END_VAR
VAR (* helpers for the ST form of the networks *)
	_t186 : BOOL;
	_t180 : BOOL;
END_VAR
(*-------------------------------------------------------------------------------------------------ПЛАНОВАЯ ПЕРЕЗАГРУЗКА МОДЕМА*)
IF MODEM_PLANOVUY_REBOOT THEN
	TIMER_DAY(IN:=TRUE, PT:=REAL_TO_TIME(TIME_PLANOVAYA_REBBOT_MODEM*60000) );
	IF TIMER_DAY.ET=TIMER_DAY.PT AND (STEP_MAIN=10 OR STEP_MAIN=520)   THEN
		IF STEP_MAIN=10 THEN
			STEP_MAIN:=600;
			TIMER_DAY(IN:=FALSE, PT:=T#0s );
			TIMER_DAY;
		END_IF
		IF STEP_MAIN=520 THEN
			STEP_MAIN:=700;
			TIMER_DAY(IN:=FALSE, PT:=T#0s );
			TIMER_DAY;
		END_IF
	END_IF
ELSE
	TIMER_DAY(IN:=FALSE, PT:=T#0s );
	TIMER_DAY;
END_IF
(*-----------------------------------------------ПЛАНОВАЯ МОДЕМА ЕСЛИ СЕРВЕР НЕ ОТВЕТИЛ БОЛЬШЕ 10 МИНУТ (НАПРИМЕР)*)
IF MODEM_WATCH_DOG THEN
	TIMER_SEND_OK(IN:=TRUE, PT:=REAL_TO_TIME(TIME_WATCH_DOG*1000));
	IF TIMER_SEND_OK.ET=TIMER_SEND_OK.PT AND (STEP_MAIN=10 OR STEP_MAIN=520)   THEN
		IF STEP_MAIN=10 THEN
			STEP_MAIN:=600;
			TIMER_SEND_OK(IN:=FALSE, PT:=T#0s );
			TIMER_SEND_OK;
		END_IF
		IF STEP_MAIN=520 THEN
			STEP_MAIN:=700;
			TIMER_SEND_OK(IN:=FALSE, PT:=T#0s );
			TIMER_SEND_OK;
		END_IF
	END_IF


	FIND_TIMER_SEND_OK:=FIND(OTVET, STRING_SEND_OK);
	IF FIND_TIMER_SEND_OK<>0 THEN
		TIMER_SEND_OK(IN:=FALSE, PT:=T#0s );
		TIMER_SEND_OK;
	END_IF
ELSE
	TIMER_SEND_OK(IN:=FALSE, PT:=T#0s );
	TIMER_SEND_OK;
END_IF

(*--------------------------------------------------------------------------------------------------ПЕРЕЗАГРУЗКА МОДЕМА С КНОПКИ*)
IF REBOOT_MODEM_SP_307 THEN
	IF STEP_MAIN=10 THEN
		STEP_MAIN:=600;
		TIMER_DAY(IN:=FALSE, PT:=T#0s );
		TIMER_DAY;
	END_IF
	IF STEP_MAIN=520 THEN
		STEP_MAIN:=700;
		TIMER_DAY(IN:=FALSE, PT:=T#0s );
		TIMER_DAY;
	END_IF
	REBOOT_MODEM_SP_307:=FALSE;
END_IF
(*--------------------------------------------------------------------------------СЛУШАЕМ ПОРТ, ЗАПИСЫВАЕМ ЗНАЧЕНИЯ В ОТВЕТ*)
P:=GetByte(0);
OTVET:=CONCAT(OTVET,RBDATA_TO_STRING(p));
IF LEN(OTVET)>255 THEN
	OTVET:='';
END_IF

(*-----------------------------------------------------------------------------------------------------------ПЕРЕЗАГРУЗКА С КНОПКИ'*)
IF REBOOT_MODEM_SP_307
THEN
	STEP_MAIN:=600;
	REBOOT_MODEM_SP_307:=FALSE;
	TIMER_REBOOT(IN:=FALSE, PT:=T#0s );
	TIMER_REBOOT;
END_IF

(*----------------------------------------------------------------------------------------------------------------ТЕСТ ОТПРАВКИ СМС'*)
IF TEST_OTPRAVKI_SMS_SP_307
THEN
	STEP_MAIN:=500;
	TEST_OTPRAVKI_SMS_SP_307:=FALSE;
	TIMER_REBOOT(IN:=FALSE, PT:=T#0s );
	TIMER_REBOOT;
END_IF
(*------------------------------------------------------------------ПЕРЕЗАГРУЗКА ПО КОЛИЧЕСТВУ ПОПЫТОК С ОТВЕТОМ ERROR'*)
IF POPUTKA>500 AND STEP_MAIN=10
THEN
	STEP_MAIN:=600;
	TIMER_REBOOT(IN:=FALSE, PT:=T#0s );
	TIMER_REBOOT;
END_IF
(*--------------------------------------------------------------------------ПЕРЕЗАГРУЗКА ПО КОЛИЧЕСТВУ ПОПЫТОК ПО ВРЕМЕНИ*)
IF POPUTKA_PO_VREMENI>6 AND STEP_MAIN=10
THEN
	STEP_MAIN:=600;
	TIMER_REBOOT(IN:=FALSE, PT:=T#0s );
	TIMER_REBOOT;
END_IF
(*------------------------------------------------------------------ПЕРЕЗАГРУЗКА ПО КОЛИЧЕСТВУ ПОПЫТОК С ОТВЕТОМ ERROR'*)
IF POPUTKA_AVARIA>400 AND STEP_MAIN=520
THEN
	STEP_MAIN:=700;
	TIMER_REBOOT(IN:=FALSE, PT:=T#0s );
	TIMER_REBOOT;
END_IF
(*-------------------------------------------------------------------------ПЕРЕЗАГРУЗКА ПО КОЛИЧЕСТВУ ПОПЫТОК ПО ВРЕМЕНИ*)
IF POPUTKA_PO_VREMENI_AVARIA>6 AND STEP_MAIN=520
THEN
	STEP_MAIN:=700;
	TIMER_REBOOT(IN:=FALSE, PT:=T#0s );
	TIMER_REBOOT;
END_IF
(*-------------------------------------------------------------------------------------------------------------ОТПРАВКА СМС АВАРИИ*)
MODEM_SOOBSHENIE_AVARIA;
	IF AVAR_SMS AND STEP_MAIN=10 AND PUSK_SP_307 THEN
		STEP_MAIN:=500;
	END_IF
(*-------------------------------------------------------------------------------------------------ОСНОВНОЙ ЦИКЛ РАБОТЫ МОДЕМА*)
CASE STEP_MAIN OF
0:
	TIMER_REBOOT(IN:=FALSE, PT:=T#0s );
	TIMER_REBOOT;
	MODEM1_ON:=TRUE;
	TIMER_ZADERGKA_OTPRAVKI_SOOBSHENIY(IN:=FALSE, PT:=T#0s );
	TIMER_ZADERGKA_OTPRAVKI_SOOBSHENIY;
	STEP_MAIN:=10;
(*---------------------------------------------------------------------------------------------------ОТПРАВКА СООБЩЕНИЙ ПО GPRS*)
10:
	MODEM_GPRS;
(*---------------------------------------------------------------------------------------------------------ОТПРАВКА АВАРИЙ ПО СМС*)
500:
	SMS_MODEM_1:=0;
	POPUTKA_AVARIA:=0;
	POPUTKA_PO_VREMENI_AVARIA:=0;
	OTVET:='';
	STEP_AVARIA:=0;
	STEP_INTO:=0;
	TIMER_ZADERGKA_OTPRAVKI_SOOBSHENIY(IN:=FALSE, PT:=T#0s );
	TIMER_ZADERGKA_OTPRAVKI_SOOBSHENIY;
	STEP_MAIN:=520;
520:
	MODEM_SMS_AVARIA;
(*--------------------------------------------------------------------------------------------------------------ПЕРЕЗАГРУЗКА МОДЕМА*)
600:
	MODEM1_ON:=FALSE;
	TIMER_REBOOT(IN:=TRUE, PT:=t#2S );
	IF TIMER_REBOOT.ET=TIMER_REBOOT.PT THEN
		STEP_MAIN:=601;
	END_IF
601:
	POPUTKA:=0;
	POPUTKA_PO_VREMENI:=0;
	REBOOT:=REBOOT+1;
	OTVET:='';
	STEP_MAIN:=0;
	STEP_MODEM:=0;
	STEP_INTO:=0;
(*-------------------------------------------------------------------------------------ПЕРЕЗАГРУЗКА МОДЕМА БЕЗ СБРОСА АВАРИИ*)
700:
	MODEM1_ON:=FALSE;
	TIMER_REBOOT(IN:=TRUE, PT:=t#2S );
	IF TIMER_REBOOT.ET=TIMER_REBOOT.PT THEN
		STEP_MAIN:=701;
	END_IF
701:
	POPUTKA:=0;
	POPUTKA_PO_VREMENI:=0;
	POPUTKA_AVARIA:=0;
	POPUTKA_PO_VREMENI_AVARIA:=0;
	REBOOT:=REBOOT+1;
	OTVET:='';
	STEP_MODEM:=0;
	STEP_AVARIA:=0;
	STEP_INTO:=0;
	POPUTKA_POSLE_REBOOT:=POPUTKA_POSLE_REBOOT+1;
	IF POPUTKA_POSLE_REBOOT>=2 THEN
		STEP_MAIN:=0;
		POPUTKA_POSLE_REBOOT:=0;
	ELSE
		STEP_MAIN:=500;
	END_IF
END_CASE
END_PROGRAM
ACTION COMMAND_AT_CGATT:
(*-----------------------------AT+CGATT? ПРОВЕРКА РЕГИСТРАЦИИ В СЕТИ ЕСЛИ 1 ТО ПЕРЕСКАКИВАЕМ ПОДКЛЮЧЕНИЕ GPRS*)
CASE STEP_INTO OF
		0:
			STR_OK:='';
			STR_ERROR:='';
			OTVET:='';
			COMMAND:='';
			STEP_INTO:=1;
			TIMER_OTVET(IN:=FALSE, PT:=T#0s );
			TIMER_OTVET;
			PAUSA(IN:=FALSE, PT:=T#0s );
			PAUSA;
		1:
			COMMAND:='AT+CGATT?';(*<-------------------------------------------------------------------------------AT-КОМАНДА*)
			STR_OK:='+CGATT: 1$R$N$R$NOK'; (*<------------------------------------------------------------ПРАВИЛЬНЫЙ ОТВЕТ*)
			STR_ERROR:='+CGATT: 0$R$N$R$NOK'; (*<-----------------------------------------------------НЕПРАВИЛЬНЫЙ ОТВЕТ*)
			COMMAND:=CONCAT(COMMAND,'$R$N');
			SetByte(0,COMMAND,LEN(COMMAND));
			STEP_INTO:=2;
		2:
			FIND_OK:=FIND(OTVET, STR_OK);
			FIND_ERROR:=FIND(OTVET, STR_ERROR);

			IF FIND_OK<>0 THEN
				PAUSA(IN:=TRUE, PT:=ZADERGKA_PEREHODA );
				IF PAUSA.ET=PAUSA.PT THEN
					STEP_MODEM:=10;(*<-------------ПЕРЕХОД К СЛЕДУЮЩЕЙ КОМАНДЕ ЕСЛИ ОТВЕТ ПОЛОЖИТЕЛЬНЫЙ*)(*10*)
					STEP_INTO:=0;
					POPUTKA:=0;
					POPUTKA_PO_VREMENI:=0;
				END_IF
			END_IF
			IF FIND_ERROR<>0 THEN
				STEP_INTO:=0;
				STEP_MODEM:=1;
				POPUTKA:=POPUTKA+1;
			END_IF
			TIMER_OTVET(IN:=TRUE, PT:=OGIDANIE_OTVETA );
			IF TIMER_OTVET.ET=TIMER_OTVET.PT THEN
				STEP_INTO:=0;
				STEP_MODEM:=190;(*<-----------------------ПЕРЕХОДИМ НА ПОСЛЕДНИЙ ШАГ ЗАКРЫТИЕ СОЕДИНЕНИЯ*)(*190*)
				POPUTKA_PO_VREMENI:=POPUTKA_PO_VREMENI+1;
				TIMER_OTVET(IN:=FALSE, PT:=T#0s );
				TIMER_OTVET;
			END_IF
END_CASE
END_ACTION
ACTION COMMAND_AT_CIFSR:
(*---------------------------------------------------------------------------------------AT+CIFSR ПОДКЛЮЧАЕМ ЛОКАЛЬНЫЙ АДРЕС*)
CASE STEP_INTO OF
		0:
			STR_OK:='';
			STR_ERROR:='';
			OTVET:='';
			COMMAND:='';
			STEP_INTO:=1;
			TIMER_OTVET(IN:=FALSE, PT:=T#0s );
			TIMER_OTVET;
			PAUSA(IN:=FALSE, PT:=T#0s );
			PAUSA;
		1:
			COMMAND:='AT+CIFSR';(*<---------------------------------------------------------------------------------AT-КОМАНДА*)
			STR_OK:='.';(*<---------------------------------------------------------------------------------------ПРАВИЛЬНЫЙ ОТВЕТ*)
			STR_ERROR:='ERROR';(*<-------------------------------------------------------------------------НЕПРАВИЛЬНЫЙ ОТВЕТ*)
			COMMAND:=CONCAT(COMMAND,'$R$N');
			SetByte(0,COMMAND,LEN(COMMAND));
			STEP_INTO:=2;
		2:
			PAUSA(IN:=TRUE, PT:=T#1S ); (*-----------------------------------ЗАПУСКАЕМ ТАЙМЕР ПАУЗА ЧТО БЫ ПОЛУЧИТЬ IP*)
			IF PAUSA.ET=PAUSA.PT THEN
				STEP_INTO:=3;
			END_IF
		3:
			FIND_OK:=FIND(OTVET, STR_OK);
			FIND_ERROR:=FIND(OTVET, STR_ERROR);

			IF FIND_OK<>0 THEN
				STEP_MODEM:=60;(*<-----------------------------------------------------ПЕРЕХОД К СЛЕДУЮЩЕЙ КОМАНДЕ*)(*60*)
				STEP_INTO:=0;
				POPUTKA:=0;
				POPUTKA_PO_VREMENI:=0;
			END_IF
			IF FIND_ERROR<>0 THEN
				STEP_MODEM:=1;
				STEP_INTO:=0;
				POPUTKA:=POPUTKA+1;
			END_IF
			TIMER_OTVET(IN:=TRUE, PT:=OGIDANIE_OTVETA );
			IF TIMER_OTVET.ET=TIMER_OTVET.PT THEN
				STEP_INTO:=0;
				STEP_MODEM:=190;(*<-----------------------ПЕРЕХОДИМ НА ПОСЛЕДНИЙ ШАГ ЗАКРЫТИЕ СОЕДИНЕНИЯ*)(*190*)
				POPUTKA_PO_VREMENI:=POPUTKA_PO_VREMENI+1;
				TIMER_OTVET(IN:=FALSE, PT:=T#0s );
				TIMER_OTVET;
			END_IF
END_CASE
END_ACTION
ACTION COMMAND_AT_CIICR:
(*-------------------------------------------------------------------------------------------------------AT+CIICR ПОДКЛЮЧАЕМ GPRS*)
CASE STEP_INTO OF
		0:
			STR_OK:='';
			STR_ERROR:='';
			OTVET:='';
			COMMAND:='';
			STEP_INTO:=1;
			TIMER_OTVET(IN:=FALSE, PT:=T#0s );
			TIMER_OTVET;
			PAUSA(IN:=FALSE, PT:=T#0s );
			PAUSA;
		1:
			COMMAND:='AT+CIICR';(*<---------------------------------------------------------------------------------AT-КОМАНДА*)
			STR_OK:='OK';(*<------------------------------------------------------------------------------------ПРАВИЛЬНЫЙ ОТВЕТ*)
			STR_ERROR:='ERROR';(*<-------------------------------------------------------------------------НЕПРАВИЛЬНЫЙ ОТВЕТ*)
			COMMAND:=CONCAT(COMMAND,'$R$N');
			SetByte(0,COMMAND,LEN(COMMAND));
			STEP_INTO:=2;
		2:
			FIND_OK:=FIND(OTVET, STR_OK);
			FIND_ERROR:=FIND(OTVET, STR_ERROR);

			IF FIND_OK<>0 THEN
				PAUSA(IN:=TRUE, PT:=ZADERGKA_PEREHODA );
				IF PAUSA.ET=PAUSA.PT THEN
					STEP_MODEM:=50;(*<-------------------------------------------------ПЕРЕХОД К СЛЕДУЮЩЕЙ КОМАНДЕ*)(*50*)
					STEP_INTO:=0;
					POPUTKA:=0;
					POPUTKA_PO_VREMENI:=0;
				END_IF
			END_IF
			IF FIND_ERROR<>0 THEN
				STEP_INTO:=0;
				STEP_MODEM:=1;
				POPUTKA:=POPUTKA+1;
			END_IF
			TIMER_OTVET(IN:=TRUE, PT:=OGIDANIE_OTVETA );
			IF TIMER_OTVET.ET=TIMER_OTVET.PT THEN
				STEP_INTO:=0;
				STEP_MODEM:=190;(*<-----------------------ПЕРЕХОДИМ НА ПОСЛЕДНИЙ ШАГ ЗАКРЫТИЕ СОЕДИНЕНИЯ*)(*190*)
				POPUTKA_PO_VREMENI:=POPUTKA_PO_VREMENI+1;
				TIMER_OTVET(IN:=FALSE, PT:=T#0s );
				TIMER_OTVET;
			END_IF
END_CASE
END_ACTION
ACTION COMMAND_AT_CIPSEND_1:
(*---------------------------------------------------------------------------------------AT+CIPSEND ЗАПРОС НА ПЕРЕДАЧУ ДАННЫХ*)
CASE STEP_INTO OF
		0:
			STR_OK:='';
			STR_ERROR:='';
			OTVET:='';
			COMMAND:='';
			STEP_INTO:=1;
			TIMER_OTVET(IN:=FALSE, PT:=T#0s );
			TIMER_OTVET;
			PAUSA(IN:=FALSE, PT:=T#0s );
			PAUSA;
		1:
			COMMAND:='AT+CIPSEND';(*<------------------------------------------------------------------------------AT-КОМАНДА*)
			STR_OK:='>';(*<--------------------------------------------------------------------------------------ПРАВИЛЬНЫЙ ОТВЕТ*)
			STR_ERROR:='ERROR';(*<-------------------------------------------------------------------------НЕПРАВИЛЬНЫЙ ОТВЕТ*)
			COMMAND:=CONCAT(COMMAND,'$R$N');
			SetByte(0,COMMAND,LEN(COMMAND));
			STEP_INTO:=2;
		2:
			FIND_OK:=FIND(OTVET, STR_OK);
			FIND_ERROR:=FIND(OTVET, STR_ERROR);

			IF FIND_OK<>0 THEN
				PAUSA(IN:=TRUE, PT:=ZADERGKA_PEREHODA );
				IF PAUSA.ET=PAUSA.PT THEN
					STEP_MODEM:=80;(*<-------------------------------------------------ПЕРЕХОД К СЛЕДУЮЩЕЙ КОМАНДЕ*)(*80*)
					STEP_INTO:=0;
					POPUTKA:=0;
					POPUTKA_PO_VREMENI:=0;
					OTVET:='';
				END_IF
			END_IF
			IF FIND_ERROR<>0 THEN
				STEP_INTO:=0;
				STEP_MODEM:=1;
				POPUTKA:=POPUTKA+1;
			END_IF
			TIMER_OTVET(IN:=TRUE, PT:=OGIDANIE_OTVETA );
			IF TIMER_OTVET.ET=TIMER_OTVET.PT THEN
				STEP_INTO:=0;
				STEP_MODEM:=190;(*<-----------------------ПЕРЕХОДИМ НА ПОСЛЕДНИЙ ШАГ ЗАКРЫТИЕ СОЕДИНЕНИЯ*)(*190*)
				POPUTKA_PO_VREMENI:=POPUTKA_PO_VREMENI+1;
				TIMER_OTVET(IN:=FALSE, PT:=T#0s );
				TIMER_OTVET;
			END_IF
END_CASE
END_ACTION
ACTION COMMAND_AT_CIPSEND_2:
(*-----------------------------------------------------------------------------AT+CIPSEND ЗАПРОС НА ПЕРЕДАЧУ ДАННЫХ ПАКЕТ 2*)
CASE STEP_INTO OF
		0:
			STR_OK:='';
			STR_ERROR:='';
			OTVET:='';
			COMMAND:='';
			STEP_INTO:=1;
			TIMER_OTVET(IN:=FALSE, PT:=T#0s );
			TIMER_OTVET;
			PAUSA(IN:=FALSE, PT:=T#0s );
			PAUSA;
		1:
			COMMAND:='AT+CIPSEND';(*<------------------------------------------------------------------------------AT-КОМАНДА*)
			STR_OK:='>';(*<--------------------------------------------------------------------------------------ПРАВИЛЬНЫЙ ОТВЕТ*)
			STR_ERROR:='ERROR';(*<-------------------------------------------------------------------------НЕПРАВИЛЬНЫЙ ОТВЕТ*)
			COMMAND:=CONCAT(COMMAND,'$R$N');
			SetByte(0,COMMAND,LEN(COMMAND));
			STEP_INTO:=2;
		2:
			FIND_OK:=FIND(OTVET, STR_OK);
			FIND_ERROR:=FIND(OTVET, STR_ERROR);

			IF FIND_OK<>0 THEN
				PAUSA(IN:=TRUE, PT:=ZADERGKA_PEREHODA );
				IF PAUSA.ET=PAUSA.PT THEN
					STEP_MODEM:=100;(*<----------------------------------------------ПЕРЕХОД К СЛЕДУЮЩЕЙ КОМАНДЕ*)(*100*)
					STEP_INTO:=0;
					POPUTKA:=0;
					POPUTKA_PO_VREMENI:=0;
					OTVET:='';
				END_IF
			END_IF
			IF FIND_ERROR<>0 THEN
				STEP_INTO:=0;
				STEP_MODEM:=1;
				POPUTKA:=POPUTKA+1;
			END_IF
			TIMER_OTVET(IN:=TRUE, PT:=OGIDANIE_OTVETA );
			IF TIMER_OTVET.ET=TIMER_OTVET.PT THEN
				STEP_INTO:=0;
				STEP_MODEM:=190;(*<-----------------------ПЕРЕХОДИМ НА ПОСЛЕДНИЙ ШАГ ЗАКРЫТИЕ СОЕДИНЕНИЯ*)(*190*)
				POPUTKA_PO_VREMENI:=POPUTKA_PO_VREMENI+1;
				TIMER_OTVET(IN:=FALSE, PT:=T#0s );
				TIMER_OTVET;
			END_IF
END_CASE
END_ACTION
ACTION COMMAND_AT_CIPSEND_3:
(*-----------------------------------------------------------------------------AT+CIPSEND ЗАПРОС НА ПЕРЕДАЧУ ДАННЫХ ПАКЕТ 2*)
CASE STEP_INTO OF
		0:
			STR_OK:='';
			STR_ERROR:='';
			OTVET:='';
			COMMAND:='';
			STEP_INTO:=1;
			TIMER_OTVET(IN:=FALSE, PT:=T#0s );
			TIMER_OTVET;
			PAUSA(IN:=FALSE, PT:=T#0s );
			PAUSA;
		1:
			COMMAND:='AT+CIPSEND';(*<------------------------------------------------------------------------------AT-КОМАНДА*)
			STR_OK:='>';(*<--------------------------------------------------------------------------------------ПРАВИЛЬНЫЙ ОТВЕТ*)
			STR_ERROR:='ERROR';(*<-------------------------------------------------------------------------НЕПРАВИЛЬНЫЙ ОТВЕТ*)
			COMMAND:=CONCAT(COMMAND,'$R$N');
			SetByte(0,COMMAND,LEN(COMMAND));
			STEP_INTO:=2;
		2:
			FIND_OK:=FIND(OTVET, STR_OK);
			FIND_ERROR:=FIND(OTVET, STR_ERROR);

			IF FIND_OK<>0 THEN
				PAUSA(IN:=TRUE, PT:=ZADERGKA_PEREHODA );
				IF PAUSA.ET=PAUSA.PT THEN
					STEP_MODEM:=120;(*<----------------------------------------------ПЕРЕХОД К СЛЕДУЮЩЕЙ КОМАНДЕ*)(*120*)
					STEP_INTO:=0;
					POPUTKA:=0;
					POPUTKA_PO_VREMENI:=0;
					OTVET:='';
				END_IF
			END_IF
			IF FIND_ERROR<>0 THEN
				STEP_INTO:=0;
				STEP_MODEM:=1;
				POPUTKA:=POPUTKA+1;
			END_IF
			TIMER_OTVET(IN:=TRUE, PT:=OGIDANIE_OTVETA );
			IF TIMER_OTVET.ET=TIMER_OTVET.PT THEN
				STEP_INTO:=0;
				STEP_MODEM:=190;(*<-----------------------ПЕРЕХОДИМ НА ПОСЛЕДНИЙ ШАГ ЗАКРЫТИЕ СОЕДИНЕНИЯ*)(*190*)
				POPUTKA_PO_VREMENI:=POPUTKA_PO_VREMENI+1;
				TIMER_OTVET(IN:=FALSE, PT:=T#0s );
				TIMER_OTVET;
			END_IF
END_CASE
END_ACTION
ACTION COMMAND_AT_CIPSHUT:
(*----------------------------------------------------------------------------------AT+CIPSHUT СБРОСИТЬ ВСЕ TCP ПОДКЛЮЧЕНИЯ*)
CASE STEP_INTO OF
		0:
			STR_OK:='';
			STR_ERROR:='';
			OTVET:='';
			COMMAND:='';
			STEP_INTO:=1;
			TIMER_OTVET(IN:=FALSE, PT:=T#0s );
			TIMER_OTVET;
			PAUSA(IN:=FALSE, PT:=T#0s );
			PAUSA;
		1:
			COMMAND:='AT+CIPSHUT';(*<------------------------------------------------------------------------------AT-КОМАНДА*)
			STR_OK:='SHUT OK';(*<------------------------------------------------------------------------------ПРАВИЛЬНЫЙ ОТВЕТ*)
			STR_ERROR:='ERROR';(*<-------------------------------------------------------------------------НЕПРАВИЛЬНЫЙ ОТВЕТ*)
			COMMAND:=CONCAT(COMMAND,'$R$N');
			SetByte(0,COMMAND,LEN(COMMAND));
			STEP_INTO:=2;
		2:
			FIND_OK:=FIND(OTVET, STR_OK);
			FIND_ERROR:=FIND(OTVET, STR_ERROR);

			IF FIND_OK<>0 THEN
				PAUSA(IN:=TRUE, PT:=ZADERGKA_PEREHODA );
				IF PAUSA.ET=PAUSA.PT THEN
					STEP_MODEM:=30;(*<-------------------------------------------------ПЕРЕХОД К СЛЕДУЮЩЕЙ КОМАНДЕ*)(*30*)
					STEP_INTO:=0;
					POPUTKA:=0;
					POPUTKA_PO_VREMENI:=0;
				END_IF
			END_IF
			IF FIND_ERROR<>0 THEN
				STEP_INTO:=0;
				STEP_MODEM:=1;
				POPUTKA:=POPUTKA+1;
			END_IF
			TIMER_OTVET(IN:=TRUE, PT:=OGIDANIE_OTVETA );
			IF TIMER_OTVET.ET=TIMER_OTVET.PT THEN
				STEP_INTO:=0;
				STEP_MODEM:=190;(*<-----------------------ПЕРЕХОДИМ НА ПОСЛЕДНИЙ ШАГ ЗАКРЫТИЕ СОЕДИНЕНИЯ*)(*190*)
				POPUTKA_PO_VREMENI:=POPUTKA_PO_VREMENI+1;
				TIMER_OTVET(IN:=FALSE, PT:=T#0s );
				TIMER_OTVET;
			END_IF
END_CASE
END_ACTION
ACTION COMMAND_AT_CIPSTART:
(*-------------------------------------------------AT+CIPSTART="TCP","ingavino.teplotehnika68.ru",80 ПОДКЛЮЧАЕМСЯ К СЕРВЕРУ*)
CASE STEP_INTO OF
		0:
			STR_OK:='';
			STR_ERROR:='';
			OTVET:='';
			COMMAND:='';
			STEP_INTO:=1;
			TIMER_OTVET(IN:=FALSE, PT:=T#0s );
			TIMER_OTVET;
			PAUSA(IN:=FALSE, PT:=T#0s );
			PAUSA;
		1:
			COMMAND:='AT+CIPSTART="TCP","karaul.teplotehnika68.ru",80';(*<-----------------------------------AT-КОМАНДА*)
			STR_OK:='CONNECT OK';(*<-------------------------------------------------------------------------ПРАВИЛЬНЫЙ ОТВЕТ*)
			STR_ERROR:='ERROR';(*<-------------------------------------------------------------------------НЕПРАВИЛЬНЫЙ ОТВЕТ*)
			COMMAND:=CONCAT(COMMAND,'$R$N');
			SetByte(0,COMMAND,LEN(COMMAND));
			STEP_INTO:=2;
		2:
			FIND_OK:=FIND(OTVET, STR_OK);
			FIND_ERROR:=FIND(OTVET, STR_ERROR);
			IF FIND_OK<>0 THEN
				PAUSA(IN:=TRUE, PT:=ZADERGKA_PEREHODA );
				IF PAUSA.ET=PAUSA.PT THEN
					STEP_MODEM:=70;(*<-------------------------------------------------ПЕРЕХОД К СЛЕДУЮЩЕЙ КОМАНДЕ*)(*70*)
					STEP_INTO:=0;
					POPUTKA:=0;
					POPUTKA_PO_VREMENI:=0;
					OTVET:='';
				END_IF
			END_IF
			IF FIND_ERROR<>0 THEN
				STEP_MODEM:=1;
				STEP_INTO:=0;
				POPUTKA:=POPUTKA+1;
			END_IF
			TIMER_OTVET(IN:=TRUE, PT:=OGIDANIE_OTVETA );
			IF TIMER_OTVET.ET=TIMER_OTVET.PT THEN
				STEP_INTO:=0;
				STEP_MODEM:=190;(*<-----------------------ПЕРЕХОДИМ НА ПОСЛЕДНИЙ ШАГ ЗАКРЫТИЕ СОЕДИНЕНИЯ*)(*190*)
				POPUTKA_PO_VREMENI:=POPUTKA_PO_VREMENI+1;
				TIMER_OTVET(IN:=FALSE, PT:=T#0s );
				TIMER_OTVET;
			END_IF
END_CASE
END_ACTION
ACTION COMMAND_AT_CSTT:
(*--------------------------------------------------------------AT+CSTT="internet.mts.ru","mts","mts" НАСТРОЙКА ТОЧКИ ДОСТУПА*)
CASE STEP_INTO OF
		0:
			STR_OK:='';
			STR_ERROR:='';
			OTVET:='';
			COMMAND:='';
			STEP_INTO:=1;
			TIMER_OTVET(IN:=FALSE, PT:=T#0s );
			TIMER_OTVET;
			PAUSA(IN:=FALSE, PT:=T#0s );
			PAUSA;
		1:
			COMMAND:='AT+CSTT="internet.mts.ru","mts","mts"';(*<---------------------------------------------------AT-КОМАНДА*)
			STR_OK:='OK';(*<------------------------------------------------------------------------------------ПРАВИЛЬНЫЙ ОТВЕТ*)
			STR_ERROR:='ERROR';(*<-------------------------------------------------------------------------НЕПРАВИЛЬНЫЙ ОТВЕТ*)
			COMMAND:=CONCAT(COMMAND,'$R$N');
			SetByte(0,COMMAND,LEN(COMMAND));
			STEP_INTO:=2;
		2:
			FIND_OK:=FIND(OTVET, STR_OK);
			FIND_ERROR:=FIND(OTVET, STR_ERROR);

			IF FIND_OK<>0 THEN
				PAUSA(IN:=TRUE, PT:=ZADERGKA_PEREHODA );
				IF PAUSA.ET=PAUSA.PT THEN
					STEP_MODEM:=40;(*<-------------------------------------------------ПЕРЕХОД К СЛЕДУЮЩЕЙ КОМАНДЕ*)(*40*)
					STEP_INTO:=0;
					POPUTKA:=0;
					POPUTKA_PO_VREMENI:=0;
				END_IF
			END_IF
			IF FIND_ERROR<>0 THEN
				STEP_INTO:=0;
				STEP_MODEM:=1;
				POPUTKA:=POPUTKA+1;
			END_IF
			TIMER_OTVET(IN:=TRUE, PT:=OGIDANIE_OTVETA );
			IF TIMER_OTVET.ET=TIMER_OTVET.PT THEN
				STEP_INTO:=0;
				STEP_MODEM:=190;(*<-----------------------ПЕРЕХОДИМ НА ПОСЛЕДНИЙ ШАГ ЗАКРЫТИЕ СОЕДИНЕНИЯ*)(*190*)
				POPUTKA_PO_VREMENI:=POPUTKA_PO_VREMENI+1;
				TIMER_OTVET(IN:=FALSE, PT:=T#0s );
				TIMER_OTVET;
			END_IF
END_CASE
END_ACTION
ACTION COMMAND_ATE0:
(*---------------------------------------------------------------------------------------------------------------ATE0 ОТКЛЮЧИТЬ ЭХО*)
CASE STEP_INTO OF
		0:
			STR_OK:='';
			STR_ERROR:='';
			OTVET:='';
			COMMAND:='';
			STEP_INTO:=1;
			TIMER_OTVET(IN:=FALSE, PT:=T#0s );
			TIMER_OTVET;
			PAUSA(IN:=FALSE, PT:=T#0s );
			PAUSA;
		1:
			COMMAND:='ATE0';(*<--------------------------------------------------------------------------------------AT-КОМАНДА*)
			STR_OK:='OK';(*<------------------------------------------------------------------------------------ПРАВИЛЬНЫЙ ОТВЕТ*)
			STR_ERROR:='ERROR';(*<-------------------------------------------------------------------------НЕПРАВИЛЬНЫЙ ОТВЕТ*)
			COMMAND:=CONCAT(COMMAND,'$R$N');
			SetByte(0,COMMAND,LEN(COMMAND));
			STEP_INTO:=2;
		2:
			FIND_OK:=FIND(OTVET, STR_OK);
			FIND_ERROR:=FIND(OTVET, STR_ERROR);

			IF FIND_OK<>0 THEN
				PAUSA(IN:=TRUE, PT:=ZADERGKA_PEREHODA );
				IF PAUSA.ET=PAUSA.PT THEN
					STEP_MODEM:=20;(*<-------------------------------------------------ПЕРЕХОД К СЛЕДУЮЩЕЙ КОМАНДЕ*)(*20*)
					STEP_INTO:=0;
					POPUTKA:=0;
					POPUTKA_PO_VREMENI:=0;
				END_IF
			END_IF
			IF FIND_ERROR<>0 THEN
				STEP_INTO:=0;
				STEP_MODEM:=1;
				POPUTKA:=POPUTKA+1;
			END_IF
			TIMER_OTVET(IN:=TRUE, PT:=OGIDANIE_OTVETA );
			IF TIMER_OTVET.ET=TIMER_OTVET.PT THEN
				STEP_INTO:=0;
				STEP_MODEM:=190;(*<-----------------------ПЕРЕХОДИМ НА ПОСЛЕДНИЙ ШАГ ЗАКРЫТИЕ СОЕДИНЕНИЯ*)(*190*)
				POPUTKA_PO_VREMENI:=POPUTKA_PO_VREMENI+1;
				TIMER_OTVET(IN:=FALSE, PT:=T#0s );
				TIMER_OTVET;
			END_IF
END_CASE
END_ACTION
ACTION MODEM_FORMIROVANIE_SMS_AVARII:
IF (AVARIA_OBRUV_DATCHIKA_T1_SP_307 AND AVARIA_OBRUV_DATCHIKA_T2_SP_307 AND AVARIA_OBRUV_DATCHIKA_T3_SP_307
	AND AVARIA_OBRUV_DATCHIKA_T4_SP_307 AND AVARIA_OBRUV_DATCHIKA_T5_SP_307 AND AVARIA_OBRUV_DATCHIKA_T6_SP_307
		AND AVARIA_OBRUV_DATCHIKA_T7_SP_307 AND AVARIA_OBRUV_DATCHIKA_T8_SP_307)
	OR (AVARIA_OBRUV_DATCHIKA_P1_SP_307 AND AVARIA_OBRUV_DATCHIKA_P2_SP_307 AND AVARIA_OBRUV_DATCHIKA_P3_SP_307
		AND AVARIA_OBRUV_DATCHIKA_P4_SP_307 AND AVARIA_OBRUV_DATCHIKA_P5_SP_307 AND AVARIA_OBRUV_DATCHIKA_P6_SP_307
			AND AVARIA_OBRUV_DATCHIKA_P7_SP_307) THEN

			STRING_SEND:=CONCAT(STRING_SEND,'AVARIA MODUL 1$R$N');
ELSE
			IF AVARIA_SETEVOY_NASOS_1_SP_307 THEN
				STRING_SEND:=CONCAT(STRING_SEND,'SETEVOY NASOS 1$R$N');
			END_IF
			IF AVARIA_SETEVOY_NASOS_2_SP_307 THEN
				STRING_SEND:=CONCAT(STRING_SEND,'AVAR.SETEVOY NASOS 2$R$N');
			END_IF
			IF AVARIA_VNUTR_NASOS_1_SP_307 THEN
				STRING_SEND:=CONCAT(STRING_SEND,'VNUTREN NASOS 1$R$N');
			END_IF
			IF AVARIA_VNUTR_NASOS_2_SP_307 THEN
				STRING_SEND:=CONCAT(STRING_SEND,'VNUTREN NASOS 2$R$N');
			END_IF
			IF AVARIA_GVS_NASOS_1_SP_307 THEN
				STRING_SEND:=CONCAT(STRING_SEND,'NASOS GVS 1$R$N');
			END_IF
			IF AVARIA_GVS_NASOS_2_SP_307 THEN
				STRING_SEND:=CONCAT(STRING_SEND,'NASOS GVS 2$R$N');
			END_IF
			IF AVARIA_PODPITOCHNYU_NASOS_1_SP_307 THEN
				STRING_SEND:=CONCAT(STRING_SEND,'PODPIT NASOS 1$R$N');
			END_IF
			IF AVARIA_PODPITOCHNYU_NASOS_2_SP_307 THEN
				STRING_SEND:=CONCAT(STRING_SEND,'PODPIT NASOS 2$R$N');
			END_IF
			(*IF AVARIA_LETNIY_NASOS_SP_307 THEN
				STRING_SEND:=CONCAT(STRING_SEND,'NL ');
			END_IF*)
			IF AVARIA_GORELKA_1_SP_307 THEN
				STRING_SEND:=CONCAT(STRING_SEND,'GORELKA 1$R$N');
			END_IF
			IF AVARIA_GORELKA_2_SP_307 THEN
				STRING_SEND:=CONCAT(STRING_SEND,'GORELKA 2$R$N');
			END_IF
			IF AVARIA_GORELKA_3_SP_307 THEN
				STRING_SEND:=CONCAT(STRING_SEND,'GORELKA 3$R$N');
			END_IF
			IF PREDUPREGDENIE_VKLUCHITE_GORELKU_1_SP_307 THEN
				STRING_SEND:=CONCAT(STRING_SEND,'ON_G1 ');
			END_IF
			IF PREDUPREGDENIE_VKLUCHITE_GORELKU_2_SP_307 THEN
				STRING_SEND:=CONCAT(STRING_SEND,'ON_G2 ');
			END_IF
			IF AVARIA_PHASA_SP_307 THEN
				STRING_SEND:=CONCAT(STRING_SEND,'PHASA$R$N');
			END_IF
			IF AVARIA_FIRE_SP_307 THEN
				STRING_SEND:=CONCAT(STRING_SEND,'POJAR$R$N');
			END_IF
			IF AVARIA_GAZ_SP_307 THEN
				STRING_SEND:=CONCAT(STRING_SEND,'GAS$R$N');
			END_IF
			IF AVARIA_VUSOKOE_DAVLENIE_OTOPLENIYA_SP_307 THEN
				STRING_SEND:=CONCAT(STRING_SEND,'VUSOK DAVL OTOPL$R$N');
			END_IF
			IF AVARIA_NIZKOE_DAVLENIE_OTOPLENIYA_SP_307 THEN
				STRING_SEND:=CONCAT(STRING_SEND,'NIZKOE DAVL OTOP$R$N');
			END_IF
			IF AVARIA_VUSOKOE_DAVLENIE_GVS_SP_307 THEN
				STRING_SEND:=CONCAT(STRING_SEND,'VUSOK DAVL GVS$R$N');
			END_IF
			IF AVARIA_NIZKOE_DAVLENIE_GVS_SP_307 THEN
				STRING_SEND:=CONCAT(STRING_SEND,'NIZKOE DAVL GVS$R$N');
			END_IF
			IF AVARIA_OBRUV_DATCHIKA_T1_SP_307 THEN
				STRING_SEND:=CONCAT(STRING_SEND,'OBRUV DAT T1$R$N');
			END_IF
			IF AVARIA_OBRUV_DATCHIKA_T2_SP_307 THEN
				STRING_SEND:=CONCAT(STRING_SEND,'OBRUV DAT T2$R$N');
			END_IF
			IF AVARIA_OBRUV_DATCHIKA_T3_SP_307 THEN
				STRING_SEND:=CONCAT(STRING_SEND,'OBRUV DAT T3$R$N');
			END_IF
			IF AVARIA_OBRUV_DATCHIKA_T4_SP_307 THEN
				STRING_SEND:=CONCAT(STRING_SEND,'OBRUV DAT T4$R$N');
			END_IF
			IF AVARIA_OBRUV_DATCHIKA_T5_SP_307 THEN
				STRING_SEND:=CONCAT(STRING_SEND,'OBRUV DAT T5$R$N');
			END_IF
			IF AVARIA_OBRUV_DATCHIKA_T6_SP_307 THEN
				STRING_SEND:=CONCAT(STRING_SEND,'OBRUV DAT T6$R$N');
			END_IF
			IF AVARIA_OBRUV_DATCHIKA_T7_SP_307 THEN
				STRING_SEND:=CONCAT(STRING_SEND,'OBRUV DAT T7$R$N');
			END_IF
			IF AVARIA_OBRUV_DATCHIKA_T8_SP_307 THEN
				STRING_SEND:=CONCAT(STRING_SEND,'OBRUV DAT T8$R$N');
			END_IF
			IF AVARIA_OBRUV_DATCHIKA_P1_SP_307 THEN
				STRING_SEND:=CONCAT(STRING_SEND,'OBRUV DAT D1$R$N');
			END_IF
			IF AVARIA_OBRUV_DATCHIKA_P2_SP_307 THEN
				STRING_SEND:=CONCAT(STRING_SEND,'OBRUV DAT D2$R$N');
			END_IF
			IF AVARIA_OBRUV_DATCHIKA_P3_SP_307 THEN
				STRING_SEND:=CONCAT(STRING_SEND,'OBRUV DAT D3$R$N');
			END_IF
			IF AVARIA_OBRUV_DATCHIKA_P4_SP_307 THEN
				STRING_SEND:=CONCAT(STRING_SEND,'OBRUV DAT D4$R$N');
			END_IF
			IF AVARIA_OBRUV_DATCHIKA_P5_SP_307 THEN
				STRING_SEND:=CONCAT(STRING_SEND,'OBRUV DAT D5$R$N');
			END_IF
			IF AVARIA_OBRUV_DATCHIKA_P6_SP_307 THEN
				STRING_SEND:=CONCAT(STRING_SEND,'OBRUV DAT D6$R$N');
			END_IF
			IF AVARIA_OBRUV_DATCHIKA_P7_SP_307 THEN
				STRING_SEND:=CONCAT(STRING_SEND,'OBRUV DAT D7$R$N');
			END_IF
			IF AVARIA_VUSOKAYA_TEMPERATURA_KOTEL_1_SP_307 THEN
				STRING_SEND:=CONCAT(STRING_SEND,'VUSOK TEMPER KOTEL 1$R$N');
			END_IF
			IF AVARIA_VUSOKAYA_TEMPERATURA_KOTEL_2_SP_307 THEN
				STRING_SEND:=CONCAT(STRING_SEND,'VUSOK TEMPER KOTEL 2$R$N');
			END_IF
			IF AVARIA_VUSOKAYA_TEMPERATURA_KOTEL_3_SP_307 THEN
				STRING_SEND:=CONCAT(STRING_SEND,'VUSOK TEMPER KOTEL 3$R$N');
			END_IF
			IF AVARIA_NAKOPITELNUY_BAK_SP_307 THEN
				STRING_SEND:=CONCAT(STRING_SEND,'NAKOPITELNUY  BAK$R$N');
			END_IF
END_IF
END_ACTION
ACTION MODEM_GPRS:
CASE STEP_MODEM OF
(*--------------------------------------------------------------------------------------------ЗАДЕРЖКА ПОСЛЕ ВКЛЮЧЕНИЯ МОДЕМА*)
0:
	TIMER_ZADERGKA_OTPRAVKI_SOOBSHENIY(IN:=TRUE, PT:=TIME_ZADERGKA_OTPRAVKI_SOOBSHENIY );
	IF TIMER_ZADERGKA_OTPRAVKI_SOOBSHENIY.ET=TIMER_ZADERGKA_OTPRAVKI_SOOBSHENIY.PT THEN
		STEP_MODEM:=1;
	END_IF
(*-----------------------------AT+CGATT? ПРОВЕРКА РЕГИСТРАЦИИ В СЕТИ ЕСЛИ 1 ТО ПЕРЕСКАКИВАЕМ ПОДКЛЮЧЕНИЕ GPRS*)
1:
	COMMAND_AT_CGATT;
(*---------------------------------------------------------------------------------------------------------------ATE0 ОТКЛЮЧИТЬ ЭХО*)
10:
	COMMAND_ATE0;
(*----------------------------------------------------------------------------------AT+CIPSHUT СБРОСИТЬ ВСЕ TCP ПОДКЛЮЧЕНИЯ*)
20:
	COMMAND_AT_CIPSHUT;
(*--------------------------------------------------------------AT+CSTT="internet.mts.ru","mts","mts" НАСТРОЙКА ТОЧКИ ДОСТУПА*)
30:
	COMMAND_AT_CSTT;
(*-------------------------------------------------------------------------------------------------------AT+CIICR ПОДКЛЮЧАЕМ GPRS*)
40:
	COMMAND_AT_CIICR;
(*---------------------------------------------------------------------------------------AT+CIFSR ПОДКЛЮЧАЕМ ЛОКАЛЬНЫЙ АДРЕС*)
50:
	COMMAND_AT_CIFSR;
(*-------------------------------------------------AT+CIPSTART="TCP","ingavino.teplotehnika68.ru",80 ПОДКЛЮЧАЕМСЯ К СЕРВЕРУ*)
60:
	COMMAND_AT_CIPSTART;
(*-----------------------------------------------------------------------------AT+CIPSEND ЗАПРОС НА ПЕРЕДАЧУ ДАННЫХ ПАКЕТ 1*)
70:
	COMMAND_AT_CIPSEND_1;
(*---------------------------------------------------------------------------------------------------------ПЕРЕДАЧА ДАННЫХ ПАКЕТ 1*)
80:
	SEND_DATA_1;
(*-----------------------------------------------------------------------------AT+CIPSEND ЗАПРОС НА ПЕРЕДАЧУ ДАННЫХ ПАКЕТ 2*)
90:
	COMMAND_AT_CIPSEND_2;
(*---------------------------------------------------------------------------------------------------------ПЕРЕДАЧА ДАННЫХ ПАКЕТ 2*)
100:
	SEND_DATA_2;
(*-----------------------------------------------------------------------------AT+CIPSEND ЗАПРОС НА ПЕРЕДАЧУ ДАННЫХ ПАКЕТ 3*)
110:
	COMMAND_AT_CIPSEND_3;
(*---------------------------------------------------------------------------------------------------------ПЕРЕДАЧА ДАННЫХ ПАКЕТ 3*)
120:
	SEND_DATA_3;
(*----------------------------------------------------------------------------------------------------------------------------------------------------------AT+CIPSEND запрос на передачу данных--------*)


(*----------------------------------------------------------------------------------------------------------------------------------------------------------передача данных СТАТУС 2--------*)







(*----------------------------------------------------------------------------------------------------------------------------------------------------------AT+CIPSHUT СБРОСИТЬ ВСЕ TCP ПОДКЛЮЧЕНИЯ--------*)
190:
CASE STEP_INTO OF
		0:
			STR_OK:='';
			STR_ERROR:='';
			OTVET:='';
			COMMAND:='';
			STEP_INTO:=1;
			TIMER_OTVET(IN:=FALSE, PT:=T#0s );(*ОБНУЛЯЕМ ТАЙМЕР ОЖИДАНИЯ ОТВЕТА*)
			TIMER_OTVET;
			PAUSA(IN:=FALSE, PT:=T#0s );(*ОБНУЛЯЕМ ТАЙМЕР ПАУЗЫ ПЕРЕД СЛЕДУЮЩЕЙ КОМАНДОЙ*)
			PAUSA;
			SetByte(0,'$0D$0A$0D$0A$1A',6);
			SetByte(0,'$0D$0A$0D$0A$1B',6);
			SetByte(0,'$0D$0A',4);

		1:
			COMMAND:='AT+CIPSHUT';(*<---------------------AT-КОМАНДА*)
			STR_OK:='SHUT OK';(*<-----------------------------------ПРАВИЛЬНЫЙ ОТВЕТ*)
			STR_ERROR:='ERROR';(*<---------------------------НЕПРАВИЛЬНЫЙ ОТВЕТ*)
			COMMAND:=CONCAT(COMMAND,'$R$N');
			SetByte(0,COMMAND,LEN(COMMAND));
			STEP_INTO:=2;
		2:
			FIND_OK:=FIND(OTVET, STR_OK);
			FIND_ERROR:=FIND(OTVET, STR_ERROR);

			IF FIND_OK<>0 THEN
				PAUSA(IN:=TRUE, PT:=(*ZADERGKA_PEREHODA*)T#1s ); (*ТАЙМЕР ЗАДЕРЖКИ ПЕРЕХОДА*)
				IF PAUSA.ET=PAUSA.PT THEN
					STEP_MODEM:=60;(*<-----------------------------ПЕРЕХОД К СЛЕДУЮЩЕЙ КОМАНДЕ*)
					STEP_INTO:=0;
					POPUTKA:=0;
					POPUTKA_PO_VREMENI:=0;
				END_IF
			END_IF
			IF FIND_ERROR<>0 THEN
				STEP_INTO:=0;
				POPUTKA:=POPUTKA+1;
			END_IF
			TIMER_OTVET(IN:=TRUE, PT:=OGIDANIE_OTVETA ); (*ЗАПУСКАЕМ ТАЙМЕР ОТВЕТА ОТ МОДЕМА ПОКА 20 СЕК*)
			IF TIMER_OTVET.ET=TIMER_OTVET.PT THEN
				STEP_INTO:=0;
				POPUTKA_PO_VREMENI:=POPUTKA_PO_VREMENI+1;
				TIMER_OTVET(IN:=FALSE, PT:=T#0s );(*ОБНУЛЯЕМ ТАЙМЕР ОЖИДАНИЯ ОТВЕТА*)
				TIMER_OTVET;
			END_IF
	END_CASE

END_CASE
END_ACTION
ACTION MODEM_OTPRAVKA_SMS_AVARII_1:
CASE STEP_AVARIA OF
(*-----------------------------------------------------------------------------------------------------ЗАДЕРЖКА ВКЛЮЧЕНИЯ МОДЕМА*)
0:
	MODEM1_ON:=TRUE;
	TIMER_ZADERGKA_OTPRAVKI_SOOBSHENIY(IN:=TRUE, PT:=T#5s );
	IF TIMER_ZADERGKA_OTPRAVKI_SOOBSHENIY.ET=TIMER_ZADERGKA_OTPRAVKI_SOOBSHENIY.PT THEN
		SetByte(0,'$R$N$R$N$1A$R$N',6);
		TIMER_OTVET(IN:=FALSE, PT:=T#0s );
		TIMER_OTVET;
		NUMBER1:='';
		NUMBER2:='';
		NUMBER3:='';
		STEP_AVARIA:=1;
	END_IF
1:
	NUMBER1:=CONCAT(NUMBER1,'+7');
	NUMBER1:=CONCAT(NUMBER1,REAL_TO_STRING(TRUNC(TEL_KOD_1)));
	NUMBER1:=CONCAT(NUMBER1,REAL_TO_STRING(TRUNC(TEL_NOMER_1)));

	NUMBER2:=CONCAT(NUMBER2,'+7');
	NUMBER2:=CONCAT(NUMBER2,REAL_TO_STRING(TRUNC(TEL_KOD_2)));
	NUMBER2:=CONCAT(NUMBER2,REAL_TO_STRING(TRUNC(TEL_NOMER_2)));

	NUMBER3:=CONCAT(NUMBER3,'+7');
	NUMBER3:=CONCAT(NUMBER3,REAL_TO_STRING(TRUNC(TEL_KOD_3)));
	NUMBER3:=CONCAT(NUMBER3,REAL_TO_STRING(TRUNC(TEL_NOMER_3)));
	NUMBER:=NUMBER1;
	STEP_AVARIA:=10;
(*----------------------------------------------------------------------------------------------------------------ATE0 ОТКЛЮЧИТЬ ЭХО*)
10:
	SMS_ATE0;
(*-----------------------------AT+CGATT? ПРОВЕРКА РЕГИСТРАЦИИ В СЕТИ ЕСЛИ 1 ТО ПЕРЕСКАКИВАЕМ ПОДКЛЮЧЕНИЕ GPRS*)
20:
	SMS_AT_CGATT;
(*---------------------------------------------------------------------------------------AT+CIPSHUT СБРОСИТЬ ВСЕ ПОДКЛЮЧЕНИЯ*)
30:
	SMS_AT_CIPSHUT;
(*----------------------------------------------------------------------------------------AT+CMGF=1 ВКЛЮЧАЕМ ТЕКСТОВЫЙ РЕЖИМ*)
40:
	SMS_AT_CMGF_1;
(*--------------------------------------------------------------------------------------------------AT+CSCS="GSM" КОДИРОВКА GSM*)
50:
	SMS_AT_CSCS_GSM;
(*---------------------------------------------------------------------------------------------------AT+CMGS="ТЕЛЕФОННЫЙ НОМЕР"*)
60:
	SMS_AT_CMGS;
(*-------------------------------------------------------------------------------------------------------------------ПЕРЕДАЧА ДАННЫХ*)
70:
	SMS_SEND_DATA;
(*--------------------------------------------------------------------------------------------------------------ВЫХОД ИЗ РЕЖИМА СМС*)
75:
	SMS_MODEM_1:=SMS_MODEM_1+1;
	IF SMS_MODEM_1>KOLICESTVO_SOOBSHENIY*KOLICHESTVO_NOMEROV-1 THEN
		STEP_MAIN:=0;
		STEP_MODEM:=1;
		NUMBER:=NUMBER1;
		TEL:=1;
	ELSE
		STEP_AVARIA:=10;
		IF TEL=1 THEN
			NUMBER:=NUMBER1;
		END_IF
		IF TEL=2 THEN
			NUMBER:=NUMBER2;
		END_IF
		IF TEL=3 THEN
			NUMBER:=NUMBER3;
		END_IF
	END_IF
END_CASE
END_ACTION
ACTION MODEM_SMS_AVARIA:
MODEM_OTPRAVKA_SMS_AVARII_1;
END_ACTION
ACTION MODEM_SOOBSHENIE_AVARIA:
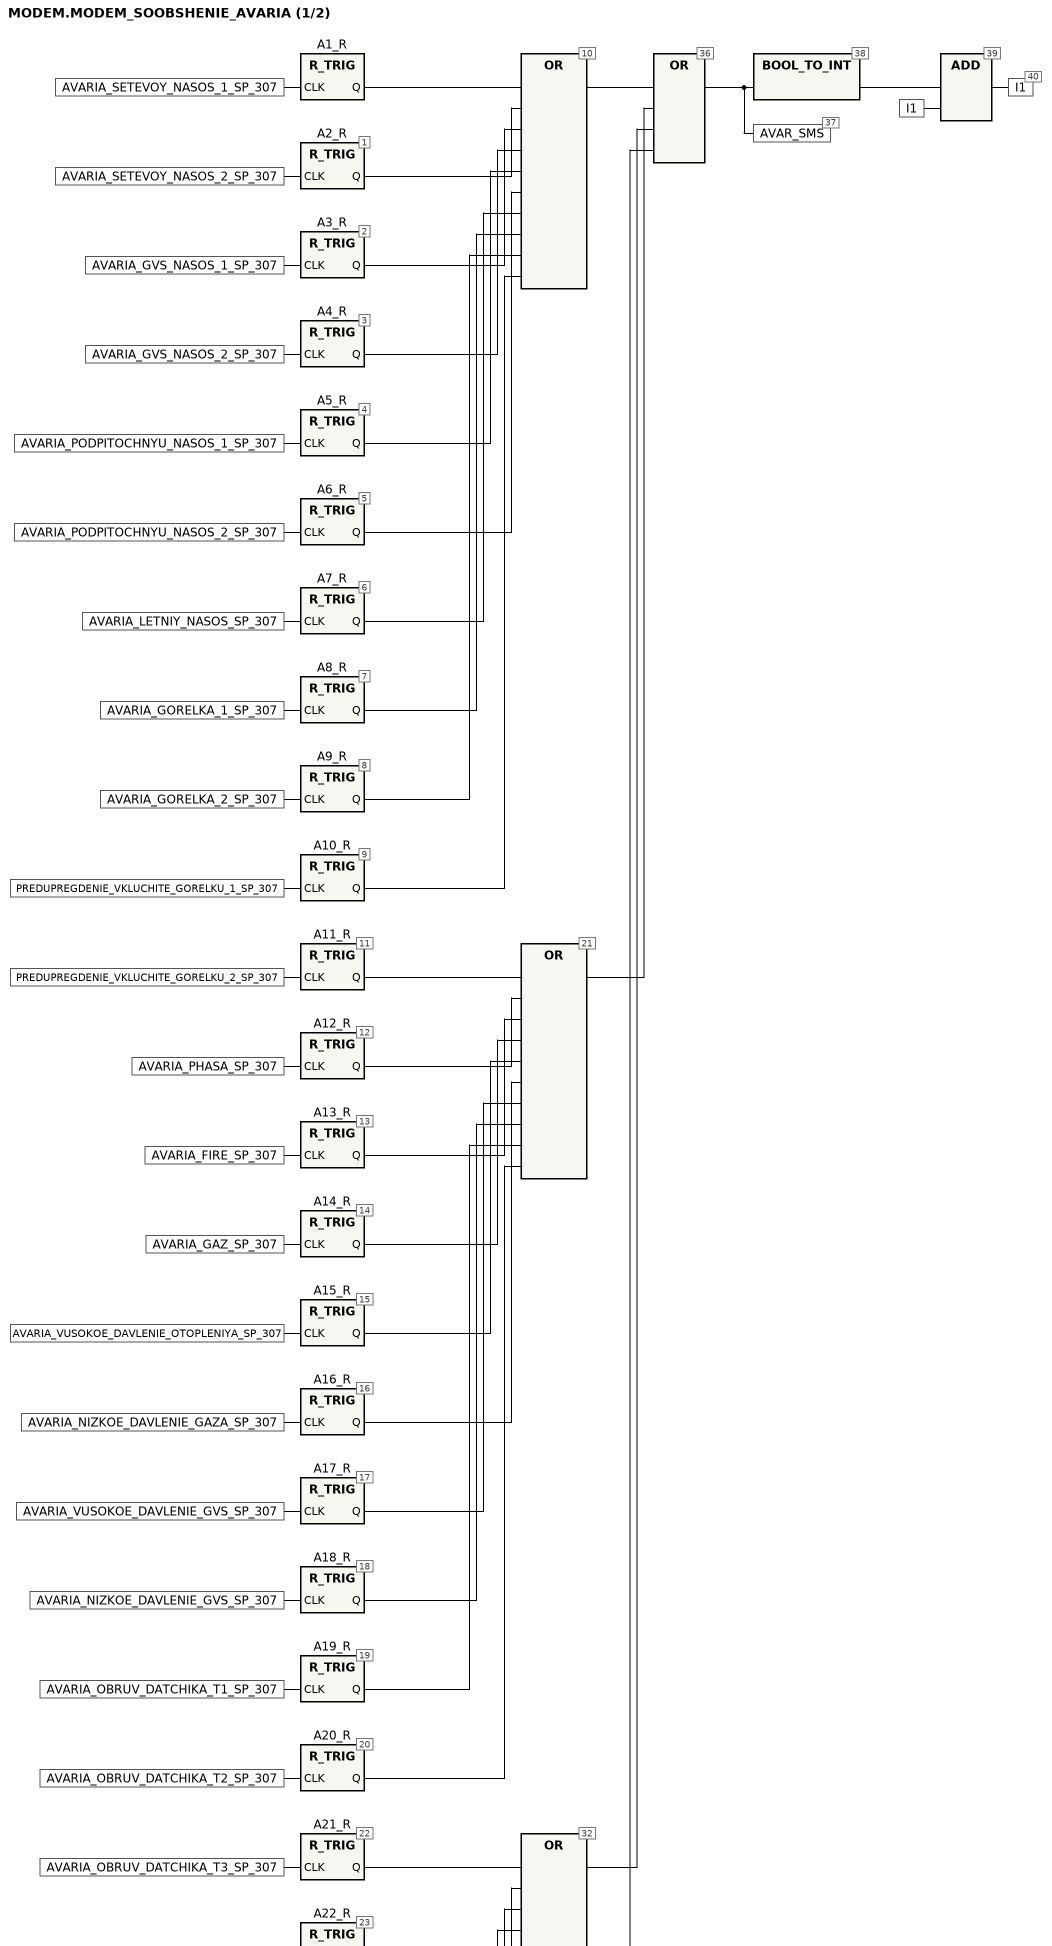
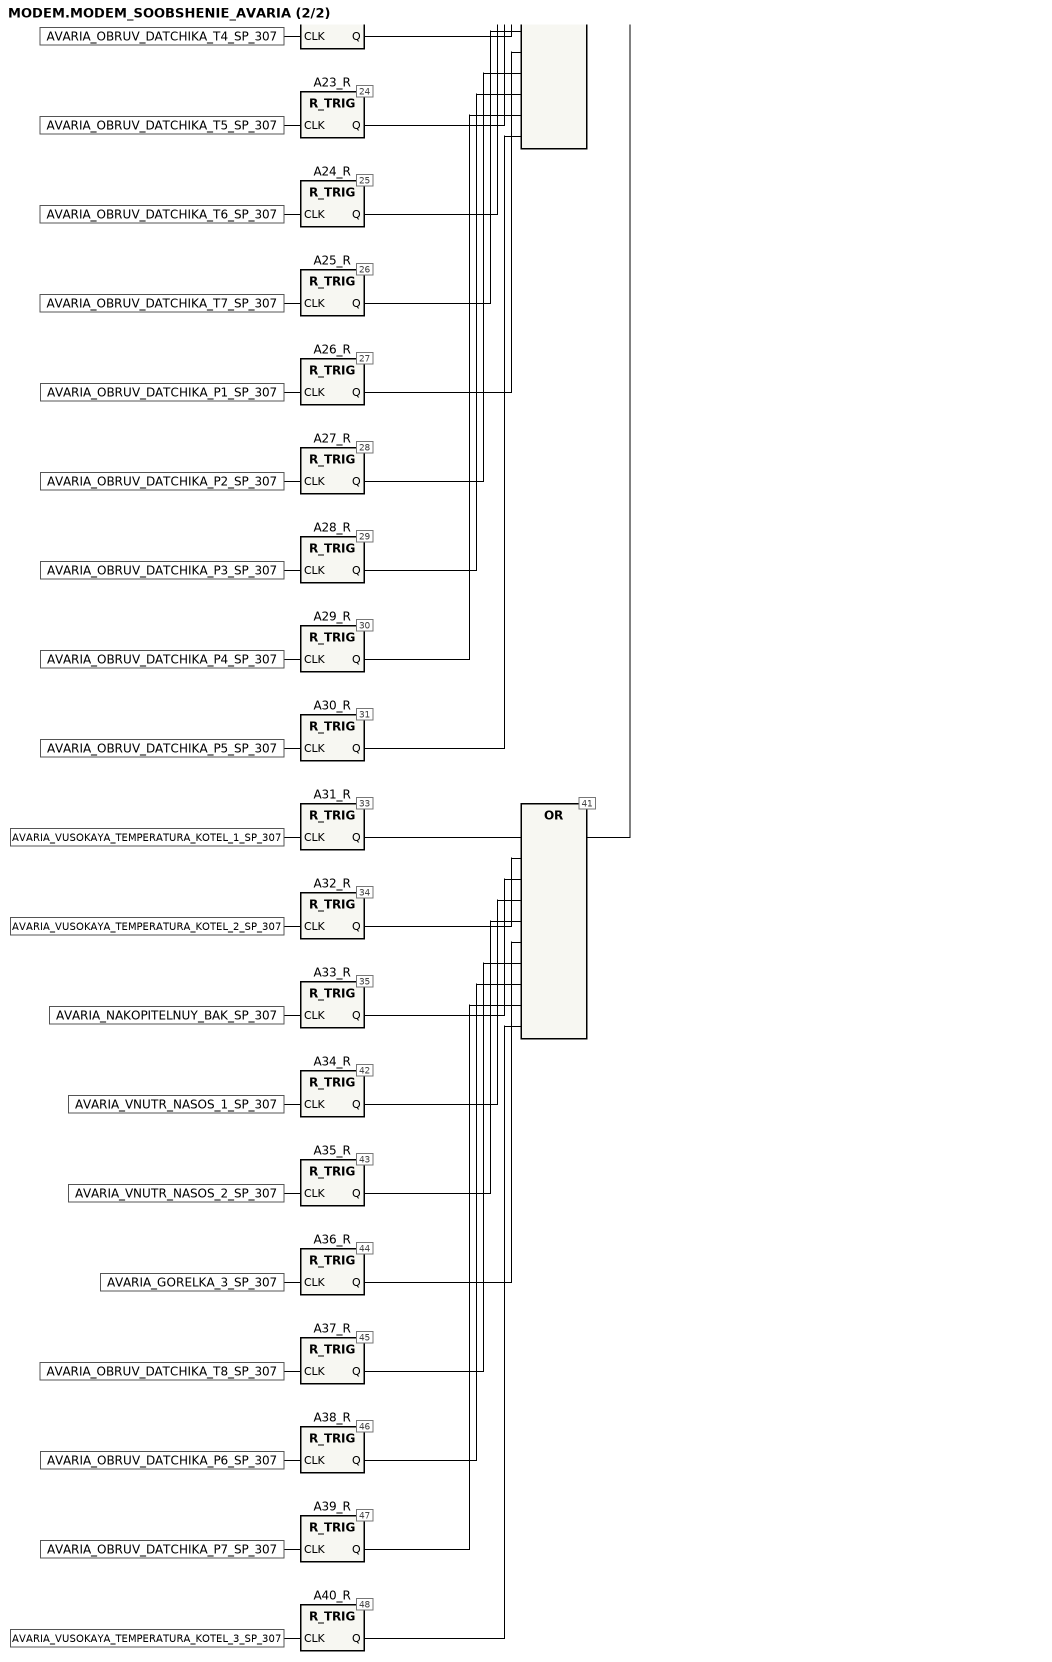
_CFC_ (* Continuous Function Chart, elements in execution order *)
#0 A1_R:R_TRIG(CLK: AVARIA_SETEVOY_NASOS_1_SP_307)
#1 A2_R:R_TRIG(CLK: AVARIA_SETEVOY_NASOS_2_SP_307)
#2 A3_R:R_TRIG(CLK: AVARIA_GVS_NASOS_1_SP_307)
#3 A4_R:R_TRIG(CLK: AVARIA_GVS_NASOS_2_SP_307)
#4 A5_R:R_TRIG(CLK: AVARIA_PODPITOCHNYU_NASOS_1_SP_307)
#5 A6_R:R_TRIG(CLK: AVARIA_PODPITOCHNYU_NASOS_2_SP_307)
#6 A7_R:R_TRIG(CLK: AVARIA_LETNIY_NASOS_SP_307)
#7 A8_R:R_TRIG(CLK: AVARIA_GORELKA_1_SP_307)
#8 A9_R:R_TRIG(CLK: AVARIA_GORELKA_2_SP_307)
#9 A10_R:R_TRIG(CLK: PREDUPREGDENIE_VKLUCHITE_GORELKU_1_SP_307)
#10 OR(#0.Q, #1.Q, #2.Q, #3.Q, #4.Q, #5.Q, #6.Q, #7.Q, #8.Q, #9.Q)
#11 A11_R:R_TRIG(CLK: PREDUPREGDENIE_VKLUCHITE_GORELKU_2_SP_307)
#12 A12_R:R_TRIG(CLK: AVARIA_PHASA_SP_307)
#13 A13_R:R_TRIG(CLK: AVARIA_FIRE_SP_307)
#14 A14_R:R_TRIG(CLK: AVARIA_GAZ_SP_307)
#15 A15_R:R_TRIG(CLK: AVARIA_VUSOKOE_DAVLENIE_OTOPLENIYA_SP_307)
#16 A16_R:R_TRIG(CLK: AVARIA_NIZKOE_DAVLENIE_GAZA_SP_307)
#17 A17_R:R_TRIG(CLK: AVARIA_VUSOKOE_DAVLENIE_GVS_SP_307)
#18 A18_R:R_TRIG(CLK: AVARIA_NIZKOE_DAVLENIE_GVS_SP_307)
#19 A19_R:R_TRIG(CLK: AVARIA_OBRUV_DATCHIKA_T1_SP_307)
#20 A20_R:R_TRIG(CLK: AVARIA_OBRUV_DATCHIKA_T2_SP_307)
#21 OR(#11.Q, #12.Q, #13.Q, #14.Q, #15.Q, #16.Q, #17.Q, #18.Q, #19.Q, #20.Q)
#22 A21_R:R_TRIG(CLK: AVARIA_OBRUV_DATCHIKA_T3_SP_307)
#23 A22_R:R_TRIG(CLK: AVARIA_OBRUV_DATCHIKA_T4_SP_307)
#24 A23_R:R_TRIG(CLK: AVARIA_OBRUV_DATCHIKA_T5_SP_307)
#25 A24_R:R_TRIG(CLK: AVARIA_OBRUV_DATCHIKA_T6_SP_307)
#26 A25_R:R_TRIG(CLK: AVARIA_OBRUV_DATCHIKA_T7_SP_307)
#27 A26_R:R_TRIG(CLK: AVARIA_OBRUV_DATCHIKA_P1_SP_307)
#28 A27_R:R_TRIG(CLK: AVARIA_OBRUV_DATCHIKA_P2_SP_307)
#29 A28_R:R_TRIG(CLK: AVARIA_OBRUV_DATCHIKA_P3_SP_307)
#30 A29_R:R_TRIG(CLK: AVARIA_OBRUV_DATCHIKA_P4_SP_307)
#31 A30_R:R_TRIG(CLK: AVARIA_OBRUV_DATCHIKA_P5_SP_307)
#32 OR(#22.Q, #23.Q, #24.Q, #25.Q, #26.Q, #27.Q, #28.Q, #29.Q, #30.Q, #31.Q)
#33 A31_R:R_TRIG(CLK: AVARIA_VUSOKAYA_TEMPERATURA_KOTEL_1_SP_307)
#34 A32_R:R_TRIG(CLK: AVARIA_VUSOKAYA_TEMPERATURA_KOTEL_2_SP_307)
#35 A33_R:R_TRIG(CLK: AVARIA_NAKOPITELNUY_BAK_SP_307)
#36 OR(#10, #21, #32, #41)
#37 AVAR_SMS <= #36
#38 BOOL_TO_INT(#36)
#39 ADD(#38, I1)
#40 I1 <= #39
#41 OR(#33.Q, #34.Q, #35.Q, #42.Q, #43.Q, #44.Q, #45.Q, #46.Q, #47.Q, #48.Q)
#42 A34_R:R_TRIG(CLK: AVARIA_VNUTR_NASOS_1_SP_307)
#43 A35_R:R_TRIG(CLK: AVARIA_VNUTR_NASOS_2_SP_307)
#44 A36_R:R_TRIG(CLK: AVARIA_GORELKA_3_SP_307)
#45 A37_R:R_TRIG(CLK: AVARIA_OBRUV_DATCHIKA_T8_SP_307)
#46 A38_R:R_TRIG(CLK: AVARIA_OBRUV_DATCHIKA_P6_SP_307)
#47 A39_R:R_TRIG(CLK: AVARIA_OBRUV_DATCHIKA_P7_SP_307)
#48 A40_R:R_TRIG(CLK: AVARIA_VUSOKAYA_TEMPERATURA_KOTEL_3_SP_307)
_END_CFC_
(* the same logic as Structured Text *)
A1_R(CLK := AVARIA_SETEVOY_NASOS_1_SP_307);
A2_R(CLK := AVARIA_SETEVOY_NASOS_2_SP_307);
A3_R(CLK := AVARIA_GVS_NASOS_1_SP_307);
A4_R(CLK := AVARIA_GVS_NASOS_2_SP_307);
A5_R(CLK := AVARIA_PODPITOCHNYU_NASOS_1_SP_307);
A6_R(CLK := AVARIA_PODPITOCHNYU_NASOS_2_SP_307);
A7_R(CLK := AVARIA_LETNIY_NASOS_SP_307);
A8_R(CLK := AVARIA_GORELKA_1_SP_307);
A9_R(CLK := AVARIA_GORELKA_2_SP_307);
A10_R(CLK := PREDUPREGDENIE_VKLUCHITE_GORELKU_1_SP_307);
A11_R(CLK := PREDUPREGDENIE_VKLUCHITE_GORELKU_2_SP_307);
A12_R(CLK := AVARIA_PHASA_SP_307);
A13_R(CLK := AVARIA_FIRE_SP_307);
A14_R(CLK := AVARIA_GAZ_SP_307);
A15_R(CLK := AVARIA_VUSOKOE_DAVLENIE_OTOPLENIYA_SP_307);
A16_R(CLK := AVARIA_NIZKOE_DAVLENIE_GAZA_SP_307);
A17_R(CLK := AVARIA_VUSOKOE_DAVLENIE_GVS_SP_307);
A18_R(CLK := AVARIA_NIZKOE_DAVLENIE_GVS_SP_307);
A19_R(CLK := AVARIA_OBRUV_DATCHIKA_T1_SP_307);
A20_R(CLK := AVARIA_OBRUV_DATCHIKA_T2_SP_307);
A21_R(CLK := AVARIA_OBRUV_DATCHIKA_T3_SP_307);
A22_R(CLK := AVARIA_OBRUV_DATCHIKA_T4_SP_307);
A23_R(CLK := AVARIA_OBRUV_DATCHIKA_T5_SP_307);
A24_R(CLK := AVARIA_OBRUV_DATCHIKA_T6_SP_307);
A25_R(CLK := AVARIA_OBRUV_DATCHIKA_T7_SP_307);
A26_R(CLK := AVARIA_OBRUV_DATCHIKA_P1_SP_307);
A27_R(CLK := AVARIA_OBRUV_DATCHIKA_P2_SP_307);
A28_R(CLK := AVARIA_OBRUV_DATCHIKA_P3_SP_307);
A29_R(CLK := AVARIA_OBRUV_DATCHIKA_P4_SP_307);
A30_R(CLK := AVARIA_OBRUV_DATCHIKA_P5_SP_307);
A31_R(CLK := AVARIA_VUSOKAYA_TEMPERATURA_KOTEL_1_SP_307);
A32_R(CLK := AVARIA_VUSOKAYA_TEMPERATURA_KOTEL_2_SP_307);
A33_R(CLK := AVARIA_NAKOPITELNUY_BAK_SP_307);
_t180 := (A1_R.Q OR A2_R.Q OR A3_R.Q OR A4_R.Q OR A5_R.Q OR A6_R.Q OR A7_R.Q OR A8_R.Q OR A9_R.Q OR A10_R.Q) OR (A11_R.Q OR A12_R.Q OR A13_R.Q OR A14_R.Q OR A15_R.Q OR A16_R.Q OR A17_R.Q OR A18_R.Q OR A19_R.Q OR A20_R.Q) OR (A21_R.Q OR A22_R.Q OR A23_R.Q OR A24_R.Q OR A25_R.Q OR A26_R.Q OR A27_R.Q OR A28_R.Q OR A29_R.Q OR A30_R.Q) OR _t186;
AVAR_SMS := _t180;
I1 := BOOL_TO_INT(_t180) + I1;
_t186 := A31_R.Q OR A32_R.Q OR A33_R.Q OR A34_R.Q OR A35_R.Q OR A36_R.Q OR A37_R.Q OR A38_R.Q OR A39_R.Q OR A40_R.Q;
A34_R(CLK := AVARIA_VNUTR_NASOS_1_SP_307);
A35_R(CLK := AVARIA_VNUTR_NASOS_2_SP_307);
A36_R(CLK := AVARIA_GORELKA_3_SP_307);
A37_R(CLK := AVARIA_OBRUV_DATCHIKA_T8_SP_307);
A38_R(CLK := AVARIA_OBRUV_DATCHIKA_P6_SP_307);
A39_R(CLK := AVARIA_OBRUV_DATCHIKA_P7_SP_307);
A40_R(CLK := AVARIA_VUSOKAYA_TEMPERATURA_KOTEL_3_SP_307);
END_ACTION
ACTION SEND_DATA_1:
(*---------------------------------------------------------------------------------------------------------ПЕРЕДАЧА ДАННЫХ ПАКЕТ 1*)
CASE STEP_INTO OF
	0:
		STR_OK:='';
		STR_ERROR:='';
		OTVET:='';
		TIMER_OTVET(IN:=FALSE, PT:=T#0s );
		TIMER_OTVET;
		PAUSA(IN:=FALSE, PT:=T#0s );
		PAUSA;

		STRING_SEND:='';
		STRING_SEND_2:='';
		STEP_INTO:=1;
	1:
		STR_OK:='SEND OK$R$NHTTP/1.1 200 OK';(*<---------------------------------------------------------ПРАВИЛЬНЫЙ ОТВЕТ*)
		STR_ERROR:='SEND OK$R$NHTTP/1.1 400 Bad Request';(*<-----------------------------------------НЕПРАВИЛЬНЫЙ ОТВЕТ*)

(*1*)		STRING_SEND_2:=CONCAT(STRING_SEND_2,'T1=');
			STRING_SEND_2:=CONCAT(STRING_SEND_2,REAL_TO_STRING(INT_TO_REAL(REAL_TO_INT(TEMPERATURA_1_PR_OTOPLENIYA_AI_SP_307*10))/10));

(*2*)		STRING_SEND_2:=CONCAT(STRING_SEND_2,'&T2=');
			STRING_SEND_2:=CONCAT(STRING_SEND_2,REAL_TO_STRING(INT_TO_REAL(REAL_TO_INT(TEMPERATURA_2_OBR_OTOPLENIYA_AI_SP_307*10))/10));

(*3*)		STRING_SEND_2:=CONCAT(STRING_SEND_2,'&T3=');
			STRING_SEND_2:=CONCAT(STRING_SEND_2,REAL_TO_STRING(INT_TO_REAL(REAL_TO_INT(TEMPERATURA_3_PR_GVS_AI_SP_307*10))/10));

(*4*)		STRING_SEND_2:=CONCAT(STRING_SEND_2,'&T4=');
			STRING_SEND_2:=CONCAT(STRING_SEND_2,REAL_TO_STRING(INT_TO_REAL(REAL_TO_INT(TEMPERATURA_4_OBR_GVS_AI_SP_307*10))/10));

(*5*)		STRING_SEND_2:=CONCAT(STRING_SEND_2,'&T5=');
			STRING_SEND_2:=CONCAT(STRING_SEND_2,REAL_TO_STRING(INT_TO_REAL(REAL_TO_INT(TEMPERATURA_5_KOTEL_1_AI_SP_307*10))/10));

(*6*)		STRING_SEND_2:=CONCAT(STRING_SEND_2,'&T6=');
			STRING_SEND_2:=CONCAT(STRING_SEND_2,REAL_TO_STRING(INT_TO_REAL(REAL_TO_INT(TEMPERATURA_6_KOTEL_2_AI_SP_307*10))/10));

(*7*)		STRING_SEND_2:=CONCAT(STRING_SEND_2,'&T7=');
			STRING_SEND_2:=CONCAT(STRING_SEND_2,REAL_TO_STRING(INT_TO_REAL(REAL_TO_INT(TEMPERATURA_7_KOTEL_3_AI_SP_307*10))/10));

(*8*)		STRING_SEND_2:=CONCAT(STRING_SEND_2,'&T8=');
			STRING_SEND_2:=CONCAT(STRING_SEND_2,REAL_TO_STRING(INT_TO_REAL(REAL_TO_INT(TEMPERATURA_8_ULICA_AI_SP_307*10))/10));

(*9*)		STRING_SEND_2:=CONCAT(STRING_SEND_2,'&D1=');
			STRING_SEND_2:=CONCAT(STRING_SEND_2,REAL_TO_STRING(INT_TO_REAL(REAL_TO_INT(DAVLENIE_1_PR_OTOPLENIYA_AI_SP_307*10))/10));

(*10*)		STRING_SEND_2:=CONCAT(STRING_SEND_2,'&D2=');
			STRING_SEND_2:=CONCAT(STRING_SEND_2,REAL_TO_STRING(INT_TO_REAL(REAL_TO_INT(DAVLENIE_2_OBR_OTOPLENIYA_AI_SP_307*10))/10));

(*11*)		STRING_SEND_2:=CONCAT(STRING_SEND_2,'&D3=');
			STRING_SEND_2:=CONCAT(STRING_SEND_2,REAL_TO_STRING(INT_TO_REAL(REAL_TO_INT(DAVLENIE_3_PR_GVS_AI_SP_307*10))/10));

(*12*)		STRING_SEND_2:=CONCAT(STRING_SEND_2,'&D4=');
			STRING_SEND_2:=CONCAT(STRING_SEND_2,REAL_TO_STRING(INT_TO_REAL(REAL_TO_INT(DAVLENIE_4_OBR_GVS_AI_SP_307*10))/10));

(*13*)		STRING_SEND_2:=CONCAT(STRING_SEND_2,'&D5=');
			STRING_SEND_2:=CONCAT(STRING_SEND_2,REAL_TO_STRING(INT_TO_REAL(REAL_TO_INT(DAVLENIE_5_PR_VNUTR_AI_SP_307*10))/10));

(*14*)		STRING_SEND_2:=CONCAT(STRING_SEND_2,'&D6=');
			STRING_SEND_2:=CONCAT(STRING_SEND_2,REAL_TO_STRING(INT_TO_REAL(REAL_TO_INT(DAVLENIE_6_OBR_VNUTR_AI_SP_307*10))/10));

(*15*)		STRING_SEND_2:=CONCAT(STRING_SEND_2,'&D7=');
			STRING_SEND_2:=CONCAT(STRING_SEND_2,REAL_TO_STRING(INT_TO_REAL(REAL_TO_INT(DAVLENIE_7_NAKOPITELNIY_BAK_AI_SP_307*10))/10));

(*16*)		STRING_SEND_2:=CONCAT(STRING_SEND_2,'&G1=');
			STRING_SEND_2:=CONCAT(STRING_SEND_2,REAL_TO_STRING(STATUS_GORELKA1_SP_307));

(*17*)		STRING_SEND_2:=CONCAT(STRING_SEND_2,'&G2=');
			STRING_SEND_2:=CONCAT(STRING_SEND_2,REAL_TO_STRING(STATUS_GORELKA2_SP_307));

(*18*)		STRING_SEND_2:=CONCAT(STRING_SEND_2,'&G3=');
			STRING_SEND_2:=CONCAT(STRING_SEND_2,REAL_TO_STRING(STATUS_GORELKA3_SP_307));



(*
		STRING_SEND_2:=CONCAT(STRING_SEND_2,'&G1P=');
		STRING_SEND_2:=CONCAT(STRING_SEND_2,REAL_TO_STRING(STATUS_GORENIE_1_B_M_SP_307));

		STRING_SEND_2:=CONCAT(STRING_SEND_2,'&G2P=');
		STRING_SEND_2:=CONCAT(STRING_SEND_2,REAL_TO_STRING(STATUS_GORENIE_2_B_M_SP_307));
*)

(*19*)		STRING_SEND_2:=CONCAT(STRING_SEND_2,'&NS1=');
			STRING_SEND_2:=CONCAT(STRING_SEND_2,REAL_TO_STRING(STATUS_NASOS_1_SETEVOY_1_SP_307));

(*20*)		STRING_SEND_2:=CONCAT(STRING_SEND_2,'&NS2=');
			STRING_SEND_2:=CONCAT(STRING_SEND_2,REAL_TO_STRING(STATUS_NASOS_2_SETEVOY_1_SP_307));

(*21*)		STRING_SEND_2:=CONCAT(STRING_SEND_2,'&SST=');
			STRING_SEND_2:=CONCAT(STRING_SEND_2,REAL_TO_STRING(STATUS_TRUBA_SETEVAYA_SP_307));

(*22*)		STRING_SEND_2:=CONCAT(STRING_SEND_2,'&NV1=');
			STRING_SEND_2:=CONCAT(STRING_SEND_2,REAL_TO_STRING(STATUS_NASOS_1_VNUTR_2_SP_307));

(*23*)		STRING_SEND_2:=CONCAT(STRING_SEND_2,'&NV2=');
			STRING_SEND_2:=CONCAT(STRING_SEND_2,REAL_TO_STRING(STATUS_NASOS_2_VNUTR_2_SP_307));

(*24*)		STRING_SEND_2:=CONCAT(STRING_SEND_2,'&SVT=');
			STRING_SEND_2:=CONCAT(STRING_SEND_2,REAL_TO_STRING(STATUS_TRUBA_VNUTR_SP_307));


(*25*)		STRING_SEND_2:=CONCAT(STRING_SEND_2,'&NG1=');
			STRING_SEND_2:=CONCAT(STRING_SEND_2,REAL_TO_STRING(STATUS_NASOS_1_GVS_3_SP_307));

(*26*)		STRING_SEND_2:=CONCAT(STRING_SEND_2,'&NG2=');
			STRING_SEND_2:=CONCAT(STRING_SEND_2,REAL_TO_STRING(STATUS_NASOS_2_GVS_3_SP_307));

(*27*)		STRING_SEND_2:=CONCAT(STRING_SEND_2,'&SGT=');
			STRING_SEND_2:=CONCAT(STRING_SEND_2,REAL_TO_STRING(STATUS_TRUBA_GVS_SP_307));

(*28*)		STRING_SEND_2:=CONCAT(STRING_SEND_2,'&NP1=');
			STRING_SEND_2:=CONCAT(STRING_SEND_2,REAL_TO_STRING(STATUS_NASOS_1_PODPIT_4_SP_307));


(*29*)		STRING_SEND_2:=CONCAT(STRING_SEND_2,'&NP2=');
			STRING_SEND_2:=CONCAT(STRING_SEND_2,REAL_TO_STRING(STATUS_NASOS_2_PODPIT_4_SP_307));

(*30*)		STRING_SEND_2:=CONCAT(STRING_SEND_2,'&SPT=');
			STRING_SEND_2:=CONCAT(STRING_SEND_2,REAL_TO_STRING(STATUS_TRUBA_PODPITKA_SP_307));

(*31*)		STRING_SEND_2:=CONCAT(STRING_SEND_2,'&NC1=');
			STRING_SEND_2:=CONCAT(STRING_SEND_2,REAL_TO_STRING(STATUS_NASOS_1_CIRCULAYCIONNUY_SP_307));

(*32*)		STRING_SEND_2:=CONCAT(STRING_SEND_2,'&NC2=');
			STRING_SEND_2:=CONCAT(STRING_SEND_2,REAL_TO_STRING(STATUS_NASOS_2_CIRCULAYCIONNUY_SP_307));

(*32*)		STRING_SEND_2:=CONCAT(STRING_SEND_2,'&NC3=');
			STRING_SEND_2:=CONCAT(STRING_SEND_2,REAL_TO_STRING(STATUS_NASOS_3_CIRCULAYCIONNUY_SP_307));

(*-----------------------------------------------------------------------------------------------------------------------------------------*)

		LEN_STRING_SEND_2:=LEN(STRING_SEND_2);(*<---------------------------------ДЛИНА ОТПРАВЛЯЕМЫХ ДАННЫХ  POST*)

		STRING_SEND:='';
		STRING_SEND:=CONCAT(STRING_SEND,'POST /index.php HTTP/1.1$0D$0A');
		STRING_SEND:=CONCAT(STRING_SEND,'Host: karaul.teplotehnika68.ru$0D$0A');
		STRING_SEND:=CONCAT(STRING_SEND,'Connection: keep-alive$0D$0A');
		STRING_SEND:=CONCAT(STRING_SEND,'Content-Type: application/x-www-form-urlencoded$0D$0A');
		STRING_SEND:=CONCAT(STRING_SEND,'Content-Length: ');
		STRING_SEND:=CONCAT(STRING_SEND,WORD_TO_STRING(LEN_STRING_SEND_2));
		STRING_SEND:=CONCAT(STRING_SEND,'$0D$0A$0D$0A');
		SetByte(0,STRING_SEND,LEN(STRING_SEND));

		SetByte(0,STRING_SEND_2,LEN(STRING_SEND_2));

		STRING_SEND:='';
		STRING_SEND:=CONCAT(STRING_SEND,'$1A');

		SetByte(0,STRING_SEND,LEN(STRING_SEND));

		OTVET:='';
		STR_FIND:=0;
		STEP_INTO:=2;
	2:
		FIND_OK:=FIND(OTVET, STR_OK);
		FIND_ERROR:=FIND(OTVET, STR_ERROR);

		IF FIND_OK<>0 THEN
			PAUSA(IN:=TRUE, PT:=ZADERGKA_PEREHODA );
			IF PAUSA.ET=PAUSA.PT THEN
				STEP_INTO:=3;
				PAUSA(IN:=FALSE, PT:=T#0s );
				PAUSA;
				POPUTKA:=0;
				POPUTKA_PO_VREMENI:=0;
				OTVET:='';
			END_IF
		END_IF
		IF FIND_ERROR<>0 THEN
			PAUSA(IN:=TRUE, PT:=ZADERGKA_PEREHODA );
			IF PAUSA.ET=PAUSA.PT THEN
				STEP_INTO:=0;
				OTVET:='';
				STEP_MODEM:=190;
			END_IF
		END_IF
		TIMER_OTVET(IN:=TRUE, PT:=OGIDANIE_OTVETA );
		IF TIMER_OTVET.ET=TIMER_OTVET.PT THEN
			STEP_INTO:=0;
			STEP_MODEM:=190;(*<---------------------------ПЕРЕХОДИМ НА ПОСЛЕДНИЙ ШАГ ЗАКРЫТИЕ СОЕДИНЕНИЯ*)(*190*)
			POPUTKA_PO_VREMENI:=POPUTKA_PO_VREMENI+1;
			TIMER_OTVET(IN:=FALSE, PT:=T#0s );
			TIMER_OTVET;
			OTVET:='';
		END_IF
	3:
		PAUSA(IN:=TRUE, PT:=ZADERGKA_PEREHODA );
		IF PAUSA.ET=PAUSA.PT THEN
			STEP_MODEM:=90;(*<---------------------------------------------------------ПЕРЕХОД К СЛЕДУЮЩЕЙ КОМАНДЕ*)(*90*)
			STEP_INTO:=0;
			POPUTKA:=0;
			POPUTKA_PO_VREMENI:=0;
		END_IF
END_CASE
END_ACTION
ACTION SEND_DATA_2:
(*---------------------------------------------------------------------------------------------------------ПЕРЕДАЧА ДАННЫХ ПАКЕТ 2*)
CASE STEP_INTO OF
	0:
		STR_OK:='';
		STR_ERROR:='';
		OTVET:='';
		TIMER_OTVET(IN:=FALSE, PT:=T#0s );
		TIMER_OTVET;
		PAUSA(IN:=FALSE, PT:=T#0s );
		PAUSA;

		STRING_SEND:='';
		STRING_SEND_2:='';
		STEP_INTO:=1;
	1:
		STR_OK:='SEND OK$R$NHTTP/1.1 200 OK';(*<---------------------------------------------------------ПРАВИЛЬНЫЙ ОТВЕТ*)
		STR_ERROR:='SEND OK$R$NHTTP/1.1 400 Bad Request';(*<-----------------------------------------НЕПРАВИЛЬНЫЙ ОТВЕТ*)

(*1*)		STRING_SEND_2:=CONCAT(STRING_SEND_2,'SSK1=');
			STRING_SEND_2:=CONCAT(STRING_SEND_2,REAL_TO_STRING(STATUS_ESBE_1_SP_307));

(*2*)		STRING_SEND_2:=CONCAT(STRING_SEND_2,'&SSK2=');
			STRING_SEND_2:=CONCAT(STRING_SEND_2,REAL_TO_STRING(STATUS_ESBE_2_SP_307));

(*3*)		STRING_SEND_2:=CONCAT(STRING_SEND_2,'&USK1=');
			STRING_SEND_2:=CONCAT(STRING_SEND_2,REAL_TO_STRING(USTAVKA_ESBE_1_SP_307));

(*4*)		STRING_SEND_2:=CONCAT(STRING_SEND_2,'&USK2=');
			STRING_SEND_2:=CONCAT(STRING_SEND_2,REAL_TO_STRING(USTAVKA_ESBE_2_SP_307));

(*5*)		STRING_SEND_2:=CONCAT(STRING_SEND_2,'&EK1=');
			STRING_SEND_2:=CONCAT(STRING_SEND_2,REAL_TO_STRING(STATUS_EL_KL_1_PODPITKA_SP_307));

(*6*)		STRING_SEND_2:=CONCAT(STRING_SEND_2,'&EK2=');
			STRING_SEND_2:=CONCAT(STRING_SEND_2,REAL_TO_STRING(STATUS_EL_KL_2_SBROS_OTOPLENIAYA_SP_307));

(*7*)		STRING_SEND_2:=CONCAT(STRING_SEND_2,'&EK3=');
			STRING_SEND_2:=CONCAT(STRING_SEND_2,REAL_TO_STRING(STATUS_EL_KL_3_SBROS_GVS_SP_307));

(*8*)		STRING_SEND_2:=CONCAT(STRING_SEND_2,'&EK4=');
			STRING_SEND_2:=CONCAT(STRING_SEND_2,REAL_TO_STRING(STATUS_EL_KL_4_NAK_BAK_SP_307));

(*9*)		STRING_SEND_2:=CONCAT(STRING_SEND_2,'&R=');
			STRING_SEND_2:=CONCAT(STRING_SEND_2,REAL_TO_STRING(REBOOT));

(*10*)		STRING_SEND_2:=CONCAT(STRING_SEND_2,'&VNS1=');
			STRING_SEND_2:=CONCAT(STRING_SEND_2,DWORD_TO_STRING(REAL_TO_DWORD(KOLICHESTVO_VKLUCHENIY_KASKAD_1_NASOS_1_SETEVOY_SP_307)));

(*11*)		STRING_SEND_2:=CONCAT(STRING_SEND_2,'&VNS2=');
			STRING_SEND_2:=CONCAT(STRING_SEND_2,DWORD_TO_STRING(REAL_TO_DWORD(KOLICHESTVO_VKLUCHENIY_KASKAD_1_NASOS_2_SETEVOY_SP_307)));

(*12*)		STRING_SEND_2:=CONCAT(STRING_SEND_2,'&VNG1=');
			STRING_SEND_2:=CONCAT(STRING_SEND_2,DWORD_TO_STRING(REAL_TO_DWORD(KOLICHESTVO_VKLUCHENIY_KASKAD_3_NASOS_1_GVS_SP_307)));

(*13*)		STRING_SEND_2:=CONCAT(STRING_SEND_2,'&VNG2=');
			STRING_SEND_2:=CONCAT(STRING_SEND_2,DWORD_TO_STRING(REAL_TO_DWORD(KOLICHESTVO_VKLUCHENIY_KASKAD_3_NASOS_2_GVS_SP_307)));

(*14*)		STRING_SEND_2:=CONCAT(STRING_SEND_2,'&VNP1=');
			STRING_SEND_2:=CONCAT(STRING_SEND_2,DWORD_TO_STRING(REAL_TO_DWORD(KOLICHESTVO_VKLUCHENIY_KASKAD_4_NASOS_1_PODPITKA_SP_307)));

(*15*)		STRING_SEND_2:=CONCAT(STRING_SEND_2,'&VNP2=');
			STRING_SEND_2:=CONCAT(STRING_SEND_2,DWORD_TO_STRING(REAL_TO_DWORD(KOLICHESTVO_VKLUCHENIY_KASKAD_4_NASOS_2_PODPITKA_SP_307)));

(*16*)		STRING_SEND_2:=CONCAT(STRING_SEND_2,'&VNV1=');
			STRING_SEND_2:=CONCAT(STRING_SEND_2,DWORD_TO_STRING(REAL_TO_DWORD(KOLICHESTVO_VKLUCHENIY_KASKAD_2_VNUTR_NASOS_1_SP_307)));

(*17*)		STRING_SEND_2:=CONCAT(STRING_SEND_2,'&VNV2=');
			STRING_SEND_2:=CONCAT(STRING_SEND_2,DWORD_TO_STRING(REAL_TO_DWORD(KOLICHESTVO_VKLUCHENIY_KASKAD_2_VNUTR_NASOS_2_SP_307)));

(*18*)		STRING_SEND_2:=CONCAT(STRING_SEND_2,'&VNC1=');
			STRING_SEND_2:=CONCAT(STRING_SEND_2,DWORD_TO_STRING(REAL_TO_DWORD(KOLICHESTVO_VKLUCHENIY_KASKAD_5_NASOS_1_CIRKUL_SP_307)));

(*19*)		STRING_SEND_2:=CONCAT(STRING_SEND_2,'&VNC2=');
			STRING_SEND_2:=CONCAT(STRING_SEND_2,DWORD_TO_STRING(REAL_TO_DWORD(KOLICHESTVO_VKLUCHENIY_KASKAD_5_NASOS_2_CIRKUL_SP_307)));

(*20*)		STRING_SEND_2:=CONCAT(STRING_SEND_2,'&VNC3=');
			STRING_SEND_2:=CONCAT(STRING_SEND_2,DWORD_TO_STRING(REAL_TO_DWORD(KOLICHESTVO_VKLUCHENIY_KASKAD_5_NASOS_3_CIRKUL_SP_307)));

(*19*)		STRING_SEND_2:=CONCAT(STRING_SEND_2,'&VG1=');
			STRING_SEND_2:=CONCAT(STRING_SEND_2,DWORD_TO_STRING(REAL_TO_DWORD(KOLICHESTVO_VKLUCHENIY_GORELKA_1_SP_307)));

(*20*)		STRING_SEND_2:=CONCAT(STRING_SEND_2,'&VG2=');
			STRING_SEND_2:=CONCAT(STRING_SEND_2,DWORD_TO_STRING(REAL_TO_DWORD(KOLICHESTVO_VKLUCHENIY_GORELKA_2_SP_307)));

(*21*)		STRING_SEND_2:=CONCAT(STRING_SEND_2,'&VG3=');
			STRING_SEND_2:=CONCAT(STRING_SEND_2,DWORD_TO_STRING(REAL_TO_DWORD(KOLICHESTVO_VKLUCHENIY_GORELKA_3_SP_307)));

(*22*)		STRING_SEND_2:=CONCAT(STRING_SEND_2,'&PNB=');
			STRING_SEND_2:=CONCAT(STRING_SEND_2,REAL_TO_STRING(STATUS_BAK_PROCENT_ZAPOLNENIA));




(*-----------------------------------------------------------------------------------------------------------------------------------------*)

		LEN_STRING_SEND_2:=LEN(STRING_SEND_2);(*<---------------------------------ДЛИНА ОТПРАВЛЯЕМЫХ ДАННЫХ  POST*)

		STRING_SEND:='';
		STRING_SEND:=CONCAT(STRING_SEND,'POST /index.php HTTP/1.1$0D$0A');
		STRING_SEND:=CONCAT(STRING_SEND,'Host: karaul.teplotehnika68.ru$0D$0A');
		STRING_SEND:=CONCAT(STRING_SEND,'Connection: keep-alive$0D$0A');
		STRING_SEND:=CONCAT(STRING_SEND,'Content-Type: application/x-www-form-urlencoded$0D$0A');
		STRING_SEND:=CONCAT(STRING_SEND,'Content-Length: ');
		STRING_SEND:=CONCAT(STRING_SEND,WORD_TO_STRING(LEN_STRING_SEND_2));
		STRING_SEND:=CONCAT(STRING_SEND,'$0D$0A$0D$0A');
		SetByte(0,STRING_SEND,LEN(STRING_SEND));

		SetByte(0,STRING_SEND_2,LEN(STRING_SEND_2));

		STRING_SEND:='';
		STRING_SEND:=CONCAT(STRING_SEND,'$1A');

		SetByte(0,STRING_SEND,LEN(STRING_SEND));

		OTVET:='';
		STR_FIND:=0;
		STEP_INTO:=2;
	2:
		FIND_OK:=FIND(OTVET, STR_OK);
		FIND_ERROR:=FIND(OTVET, STR_ERROR);

		IF FIND_OK<>0 THEN
			PAUSA(IN:=TRUE, PT:=ZADERGKA_PEREHODA );
			IF PAUSA.ET=PAUSA.PT THEN
				STEP_INTO:=3;
				PAUSA(IN:=FALSE, PT:=T#0s );
				PAUSA;
				POPUTKA:=0;
				POPUTKA_PO_VREMENI:=0;
				OTVET:='';
			END_IF
		END_IF
		IF FIND_ERROR<>0 THEN
			PAUSA(IN:=TRUE, PT:=ZADERGKA_PEREHODA );
			IF PAUSA.ET=PAUSA.PT THEN
				STEP_INTO:=0;
				OTVET:='';
				STEP_MODEM:=190;
			END_IF
		END_IF
		TIMER_OTVET(IN:=TRUE, PT:=OGIDANIE_OTVETA );
		IF TIMER_OTVET.ET=TIMER_OTVET.PT THEN
			STEP_INTO:=0;
			STEP_MODEM:=190;(*<---------------------------ПЕРЕХОДИМ НА ПОСЛЕДНИЙ ШАГ ЗАКРЫТИЕ СОЕДИНЕНИЯ*)(*190*)
			POPUTKA_PO_VREMENI:=POPUTKA_PO_VREMENI+1;
			TIMER_OTVET(IN:=FALSE, PT:=T#0s );
			TIMER_OTVET;
			OTVET:='';
		END_IF
	3:
		PAUSA(IN:=TRUE, PT:=ZADERGKA_PEREHODA );
		IF PAUSA.ET=PAUSA.PT THEN
			STEP_MODEM:=110;(*<-------------------------------------------------------ПЕРЕХОД К СЛЕДУЮЩЕЙ КОМАНДЕ*)(*110*)
			STEP_INTO:=0;
			POPUTKA:=0;
			POPUTKA_PO_VREMENI:=0;
		END_IF
END_CASE
END_ACTION
ACTION SEND_DATA_3:
(*---------------------------------------------------------------------------------------------------------ПЕРЕДАЧА ДАННЫХ ПАКЕТ 2*)
CASE STEP_INTO OF
	0:
		STR_OK:='';
		STR_ERROR:='';
		OTVET:='';
		TIMER_OTVET(IN:=FALSE, PT:=T#0s );
		TIMER_OTVET;
		PAUSA(IN:=FALSE, PT:=T#0s );
		PAUSA;

		STRING_SEND:='';
		STRING_SEND_2:='';
		STEP_INTO:=1;
	1:
		STR_OK:='SEND OK$R$NHTTP/1.1 200 OK';(*<---------------------------------------------------------ПРАВИЛЬНЫЙ ОТВЕТ*)
		STR_ERROR:='SEND OK$R$NHTTP/1.1 400 Bad Request';(*<-----------------------------------------НЕПРАВИЛЬНЫЙ ОТВЕТ*)

(*1*)		STRING_SEND_2:=CONCAT(STRING_SEND_2,'A1=');
			STRING_SEND_2:=CONCAT(STRING_SEND_2,INT_TO_STRING(BOOL_TO_INT(AVARIA_SETEVOY_NASOS_1_SP_307)));

(*2*)		STRING_SEND_2:=CONCAT(STRING_SEND_2,'&A2=');
			STRING_SEND_2:=CONCAT(STRING_SEND_2,INT_TO_STRING(BOOL_TO_INT(AVARIA_SETEVOY_NASOS_2_SP_307)));

		STRING_SEND_2:=CONCAT(STRING_SEND_2,'&A3=');
		STRING_SEND_2:=CONCAT(STRING_SEND_2,INT_TO_STRING(BOOL_TO_INT(AVARIA_GVS_NASOS_1_SP_307)));

		STRING_SEND_2:=CONCAT(STRING_SEND_2,'&A4=');
		STRING_SEND_2:=CONCAT(STRING_SEND_2,INT_TO_STRING(BOOL_TO_INT(AVARIA_GVS_NASOS_2_SP_307)));

		STRING_SEND_2:=CONCAT(STRING_SEND_2,'&A5=');
		STRING_SEND_2:=CONCAT(STRING_SEND_2,INT_TO_STRING(BOOL_TO_INT(AVARIA_PODPITOCHNYU_NASOS_1_SP_307)));

		STRING_SEND_2:=CONCAT(STRING_SEND_2,'&A6=');
		STRING_SEND_2:=CONCAT(STRING_SEND_2,INT_TO_STRING(BOOL_TO_INT(AVARIA_PODPITOCHNYU_NASOS_2_SP_307)));

		STRING_SEND_2:=CONCAT(STRING_SEND_2,'&A7=');
		STRING_SEND_2:=CONCAT(STRING_SEND_2,INT_TO_STRING(BOOL_TO_INT(AVARIA_LETNIY_NASOS_SP_307)));

		STRING_SEND_2:=CONCAT(STRING_SEND_2,'&A8=');
		STRING_SEND_2:=CONCAT(STRING_SEND_2,INT_TO_STRING(BOOL_TO_INT(AVARIA_GORELKA_1_SP_307)));

		STRING_SEND_2:=CONCAT(STRING_SEND_2,'&A9=');
		STRING_SEND_2:=CONCAT(STRING_SEND_2,INT_TO_STRING(BOOL_TO_INT(AVARIA_GORELKA_2_SP_307)));

		STRING_SEND_2:=CONCAT(STRING_SEND_2,'&A10=');
		STRING_SEND_2:=CONCAT(STRING_SEND_2,INT_TO_STRING(BOOL_TO_INT(PREDUPREGDENIE_VKLUCHITE_GORELKU_1_SP_307)));

		STRING_SEND_2:=CONCAT(STRING_SEND_2,'&A11=');
		STRING_SEND_2:=CONCAT(STRING_SEND_2,INT_TO_STRING(BOOL_TO_INT(PREDUPREGDENIE_VKLUCHITE_GORELKU_2_SP_307)));

		STRING_SEND_2:=CONCAT(STRING_SEND_2,'&A12=');
		STRING_SEND_2:=CONCAT(STRING_SEND_2,INT_TO_STRING(BOOL_TO_INT(AVARIA_PHASA_SP_307)));

		STRING_SEND_2:=CONCAT(STRING_SEND_2,'&A13=');
		STRING_SEND_2:=CONCAT(STRING_SEND_2,INT_TO_STRING(BOOL_TO_INT(AVARIA_FIRE_SP_307)));

		STRING_SEND_2:=CONCAT(STRING_SEND_2,'&A14=');
		STRING_SEND_2:=CONCAT(STRING_SEND_2,INT_TO_STRING(BOOL_TO_INT(AVARIA_GAZ_SP_307)));

		STRING_SEND_2:=CONCAT(STRING_SEND_2,'&A15=');
		STRING_SEND_2:=CONCAT(STRING_SEND_2,INT_TO_STRING(BOOL_TO_INT(AVARIA_VUSOKOE_DAVLENIE_OTOPLENIYA_SP_307)));

		STRING_SEND_2:=CONCAT(STRING_SEND_2,'&A16=');
		STRING_SEND_2:=CONCAT(STRING_SEND_2,INT_TO_STRING(BOOL_TO_INT(AVARIA_NIZKOE_DAVLENIE_OTOPLENIYA_SP_307)));

		STRING_SEND_2:=CONCAT(STRING_SEND_2,'&A17=');
		STRING_SEND_2:=CONCAT(STRING_SEND_2,INT_TO_STRING(BOOL_TO_INT(AVARIA_VUSOKOE_DAVLENIE_GVS_SP_307)));

		STRING_SEND_2:=CONCAT(STRING_SEND_2,'&A18=');
		STRING_SEND_2:=CONCAT(STRING_SEND_2,INT_TO_STRING(BOOL_TO_INT(AVARIA_NIZKOE_DAVLENIE_GVS_SP_307)));

		STRING_SEND_2:=CONCAT(STRING_SEND_2,'&A19=');
		STRING_SEND_2:=CONCAT(STRING_SEND_2,INT_TO_STRING(BOOL_TO_INT(AVARIA_OBRUV_DATCHIKA_T1_SP_307)));

		STRING_SEND_2:=CONCAT(STRING_SEND_2,'&A20=');
		STRING_SEND_2:=CONCAT(STRING_SEND_2,INT_TO_STRING(BOOL_TO_INT(AVARIA_OBRUV_DATCHIKA_T2_SP_307)));

		STRING_SEND_2:=CONCAT(STRING_SEND_2,'&A21=');
		STRING_SEND_2:=CONCAT(STRING_SEND_2,INT_TO_STRING(BOOL_TO_INT(AVARIA_OBRUV_DATCHIKA_T3_SP_307)));

		STRING_SEND_2:=CONCAT(STRING_SEND_2,'&A22=');
		STRING_SEND_2:=CONCAT(STRING_SEND_2,INT_TO_STRING(BOOL_TO_INT(AVARIA_OBRUV_DATCHIKA_T4_SP_307)));

		STRING_SEND_2:=CONCAT(STRING_SEND_2,'&A23=');
		STRING_SEND_2:=CONCAT(STRING_SEND_2,INT_TO_STRING(BOOL_TO_INT(AVARIA_OBRUV_DATCHIKA_T5_SP_307)));

		STRING_SEND_2:=CONCAT(STRING_SEND_2,'&A24=');
		STRING_SEND_2:=CONCAT(STRING_SEND_2,INT_TO_STRING(BOOL_TO_INT(AVARIA_OBRUV_DATCHIKA_T6_SP_307)));

		STRING_SEND_2:=CONCAT(STRING_SEND_2,'&A25=');
		STRING_SEND_2:=CONCAT(STRING_SEND_2,INT_TO_STRING(BOOL_TO_INT(AVARIA_OBRUV_DATCHIKA_T7_SP_307)));

		STRING_SEND_2:=CONCAT(STRING_SEND_2,'&A26=');
		STRING_SEND_2:=CONCAT(STRING_SEND_2,INT_TO_STRING(BOOL_TO_INT(AVARIA_OBRUV_DATCHIKA_P1_SP_307)));

		STRING_SEND_2:=CONCAT(STRING_SEND_2,'&A27=');
		STRING_SEND_2:=CONCAT(STRING_SEND_2,INT_TO_STRING(BOOL_TO_INT(AVARIA_OBRUV_DATCHIKA_P2_SP_307)));

		STRING_SEND_2:=CONCAT(STRING_SEND_2,'&A28=');
		STRING_SEND_2:=CONCAT(STRING_SEND_2,INT_TO_STRING(BOOL_TO_INT(AVARIA_OBRUV_DATCHIKA_P3_SP_307)));

		STRING_SEND_2:=CONCAT(STRING_SEND_2,'&A29=');
		STRING_SEND_2:=CONCAT(STRING_SEND_2,INT_TO_STRING(BOOL_TO_INT(AVARIA_OBRUV_DATCHIKA_P4_SP_307)));

		STRING_SEND_2:=CONCAT(STRING_SEND_2,'&A30=');
		STRING_SEND_2:=CONCAT(STRING_SEND_2,INT_TO_STRING(BOOL_TO_INT(AVARIA_OBRUV_DATCHIKA_P5_SP_307)));

		STRING_SEND_2:=CONCAT(STRING_SEND_2,'&A31=');
		STRING_SEND_2:=CONCAT(STRING_SEND_2,INT_TO_STRING(BOOL_TO_INT(AVARIA_VUSOKAYA_TEMPERATURA_KOTEL_1_SP_307)));

		STRING_SEND_2:=CONCAT(STRING_SEND_2,'&A32=');
		STRING_SEND_2:=CONCAT(STRING_SEND_2,INT_TO_STRING(BOOL_TO_INT(AVARIA_VUSOKAYA_TEMPERATURA_KOTEL_2_SP_307)));

		STRING_SEND_2:=CONCAT(STRING_SEND_2,'&A33=');
		STRING_SEND_2:=CONCAT(STRING_SEND_2,INT_TO_STRING(BOOL_TO_INT(AVARIA_NAKOPITELNUY_BAK_SP_307)));


(*-----------------------------------------------------------------------------------------------------------------------------------------*)

		LEN_STRING_SEND_2:=LEN(STRING_SEND_2);(*<---------------------------------ДЛИНА ОТПРАВЛЯЕМЫХ ДАННЫХ  POST*)

		STRING_SEND:='';
		STRING_SEND:=CONCAT(STRING_SEND,'POST /index.php HTTP/1.1$0D$0A');
		STRING_SEND:=CONCAT(STRING_SEND,'Host: karaul.teplotehnika68.ru$0D$0A');
		STRING_SEND:=CONCAT(STRING_SEND,'Connection: close$0D$0A');
		STRING_SEND:=CONCAT(STRING_SEND,'Content-Type: application/x-www-form-urlencoded$0D$0A');
		STRING_SEND:=CONCAT(STRING_SEND,'Content-Length: ');
		STRING_SEND:=CONCAT(STRING_SEND,WORD_TO_STRING(LEN_STRING_SEND_2));
		STRING_SEND:=CONCAT(STRING_SEND,'$0D$0A$0D$0A');
		SetByte(0,STRING_SEND,LEN(STRING_SEND));

		SetByte(0,STRING_SEND_2,LEN(STRING_SEND_2));

		STRING_SEND:='';
		STRING_SEND:=CONCAT(STRING_SEND,'$1A');

		SetByte(0,STRING_SEND,LEN(STRING_SEND));

		OTVET:='';
		STR_FIND:=0;
		STEP_INTO:=2;
	2:
		FIND_OK:=FIND(OTVET, STR_OK);
		FIND_ERROR:=FIND(OTVET, STR_ERROR);

		IF FIND_OK<>0 THEN
			PAUSA(IN:=TRUE, PT:=ZADERGKA_PEREHODA );
			IF PAUSA.ET=PAUSA.PT THEN
				STEP_INTO:=3;
				PAUSA(IN:=FALSE, PT:=T#0s );
				PAUSA;
				POPUTKA:=0;
				POPUTKA_PO_VREMENI:=0;
				OTVET:='';
			END_IF
		END_IF
		IF FIND_ERROR<>0 THEN
			PAUSA(IN:=TRUE, PT:=ZADERGKA_PEREHODA );
			IF PAUSA.ET=PAUSA.PT THEN
				STEP_INTO:=0;
				OTVET:='';
				STEP_MODEM:=190;
			END_IF
		END_IF
		TIMER_OTVET(IN:=TRUE, PT:=OGIDANIE_OTVETA );
		IF TIMER_OTVET.ET=TIMER_OTVET.PT THEN
			STEP_INTO:=0;
			STEP_MODEM:=190;(*<---------------------------ПЕРЕХОДИМ НА ПОСЛЕДНИЙ ШАГ ЗАКРЫТИЕ СОЕДИНЕНИЯ*)(*190*)
			POPUTKA_PO_VREMENI:=POPUTKA_PO_VREMENI+1;
			TIMER_OTVET(IN:=FALSE, PT:=T#0s );
			TIMER_OTVET;
			OTVET:='';
		END_IF
	3:
		PAUSA(IN:=TRUE, PT:=ZADERGKA_PEREHODA );
		IF PAUSA.ET=PAUSA.PT THEN
			STEP_MODEM:=190;(*<-------------------------------------------------------ПЕРЕХОД К СЛЕДУЮЩЕЙ КОМАНДЕ*)(*110*)
			STEP_INTO:=0;
			POPUTKA:=0;
			POPUTKA_PO_VREMENI:=0;
		END_IF
END_CASE
END_ACTION
ACTION SMS_AT_CGATT:
(*-----------------------------AT+CGATT? ПРОВЕРКА РЕГИСТРАЦИИ В СЕТИ ЕСЛИ 1 ТО ПЕРЕСКАКИВАЕМ ПОДКЛЮЧЕНИЕ GPRS*)
CASE STEP_INTO OF
		0:
			STR_OK:='';
			STR_ERROR:='';
			OTVET:='';
			COMMAND:='';
			STEP_INTO:=1;
			TIMER_OTVET(IN:=FALSE, PT:=T#0s );
			TIMER_OTVET;
			PAUSA(IN:=FALSE, PT:=T#0s );
			PAUSA;
		1:
			COMMAND:='AT+CGATT?';(*<-------------------------------------------------------------------------------AT-КОМАНДА*)
			STR_OK:='+CGATT: 1$R$N$R$NOK'; (*<------------------------------------------------------------ПРАВИЛЬНЫЙ ОТВЕТ*)
			STR_ERROR:='+CGATT: 0$R$N$R$NOK'; (*<-----------------------------------------------------НЕПРАВИЛЬНЫЙ ОТВЕТ*)
			COMMAND:=CONCAT(COMMAND,'$R$N');
			SetByte(0,COMMAND,LEN(COMMAND));
			STEP_INTO:=2;
		2:
			FIND_OK:=FIND(OTVET, STR_OK);
			FIND_ERROR:=FIND(OTVET, STR_ERROR);

			IF FIND_OK<>0 THEN
				PAUSA(IN:=TRUE, PT:=ZADERGKA_PEREHODA );
				IF PAUSA.ET=PAUSA.PT THEN
					STEP_AVARIA:=30;(*<-------------------------------------------------ПЕРЕХОД К СЛЕДУЮЩЕЙ КОМАНДЕ*)(*30*)
					STEP_INTO:=0;
					POPUTKA_AVARIA:=0;
					POPUTKA_PO_VREMENI_AVARIA:=0;
				END_IF
			END_IF
			IF FIND_ERROR<>0 THEN
				STEP_INTO:=0;
				POPUTKA_AVARIA:=POPUTKA_AVARIA+1;
			END_IF
			TIMER_OTVET(IN:=TRUE, PT:=OGIDANIE_OTVETA );
			IF TIMER_OTVET.ET=TIMER_OTVET.PT THEN
				STEP_INTO:=0;
				POPUTKA_PO_VREMENI_AVARIA:=POPUTKA_PO_VREMENI_AVARIA+1;
				TIMER_OTVET(IN:=FALSE, PT:=T#0s );
				TIMER_OTVET;
			END_IF
END_CASE
END_ACTION
ACTION SMS_AT_CIPSHUT:
(*---------------------------------------------------------------------------------------AT+CIPSHUT СБРОСИТЬ ВСЕ ПОДКЛЮЧЕНИЯ*)
CASE STEP_INTO OF
		0:
			STR_OK:='';
			STR_ERROR:='';
			OTVET:='';
			COMMAND:='';
			STEP_INTO:=1;
			TIMER_OTVET(IN:=FALSE, PT:=T#0s );
			TIMER_OTVET;
			PAUSA(IN:=FALSE, PT:=T#0s );
			PAUSA;
		1:
			COMMAND:='AT+CIPSHUT';(*<------------------------------------------------------------------------------AT-КОМАНДА*)
			STR_OK:='SHUT OK';(*<------------------------------------------------------------------------------ПРАВИЛЬНЫЙ ОТВЕТ*)
			STR_ERROR:='ERROR';(*<-------------------------------------------------------------------------НЕПРАВИЛЬНЫЙ ОТВЕТ*)
			COMMAND:=CONCAT(COMMAND,'$R$N');
			SetByte(0,COMMAND,LEN(COMMAND));
			STEP_INTO:=2;
		2:
			FIND_OK:=FIND(OTVET, STR_OK);
			FIND_ERROR:=FIND(OTVET, STR_ERROR);

			IF FIND_OK<>0 THEN
				PAUSA(IN:=TRUE, PT:=ZADERGKA_PEREHODA );
				IF PAUSA.ET=PAUSA.PT THEN
					STEP_AVARIA:=40;(*<-------------------------------------------------ПЕРЕХОД К СЛЕДУЮЩЕЙ КОМАНДЕ*)(*40*)
					STEP_INTO:=0;
					POPUTKA_AVARIA:=0;
					POPUTKA_PO_VREMENI_AVARIA:=0;
				END_IF
			END_IF
			IF FIND_ERROR<>0 THEN
				STEP_INTO:=0;
				POPUTKA_AVARIA:=POPUTKA_AVARIA+1;
			END_IF
			TIMER_OTVET(IN:=TRUE, PT:=OGIDANIE_OTVETA );
			IF TIMER_OTVET.ET=TIMER_OTVET.PT THEN
				STEP_INTO:=0;
				POPUTKA_PO_VREMENI_AVARIA:=POPUTKA_PO_VREMENI_AVARIA+1;
				TIMER_OTVET(IN:=FALSE, PT:=T#0s );
				TIMER_OTVET;
			END_IF
END_CASE
END_ACTION
ACTION SMS_AT_CMGF_1:
(*----------------------------------------------------------------------------------------AT+CMGF=1 ВКЛЮЧАЕМ ТЕКСТОВЫЙ РЕЖИМ*)
CASE STEP_INTO OF
		0:
			STR_OK:='';
			STR_ERROR:='';
			OTVET:='';
			COMMAND:='';
			STEP_INTO:=1;
			TIMER_OTVET(IN:=FALSE, PT:=T#0s );
			TIMER_OTVET;
			PAUSA(IN:=FALSE, PT:=T#0s );
			PAUSA;
		1:
			COMMAND:='AT+CMGF=1';(*<-------------------------------------------------------------------------------AT-КОМАНДА*)
			STR_OK:='OK';(*<------------------------------------------------------------------------------------ПРАВИЛЬНЫЙ ОТВЕТ*)
			STR_ERROR:='ERROR';(*<-------------------------------------------------------------------------НЕПРАВИЛЬНЫЙ ОТВЕТ*)
			COMMAND:=CONCAT(COMMAND,'$R$N');
			SetByte(0,COMMAND,LEN(COMMAND));
			STEP_INTO:=2;
		2:
			FIND_OK:=FIND(OTVET, STR_OK);
			FIND_ERROR:=FIND(OTVET, STR_ERROR);

			IF FIND_OK<>0 THEN
				PAUSA(IN:=TRUE, PT:=ZADERGKA_PEREHODA );
				IF PAUSA.ET=PAUSA.PT THEN
					STEP_AVARIA:=50;(*<-------------------------------------------------ПЕРЕХОД К СЛЕДУЮЩЕЙ КОМАНДЕ*)(*50*)
					STEP_INTO:=0;
					POPUTKA_AVARIA:=0;
					POPUTKA_PO_VREMENI_AVARIA:=0;
				END_IF
			END_IF
			IF FIND_ERROR<>0 THEN
				STEP_INTO:=0;
				POPUTKA_AVARIA:=POPUTKA_AVARIA+1;
			END_IF
			TIMER_OTVET(IN:=TRUE, PT:=OGIDANIE_OTVETA );
			IF TIMER_OTVET.ET=TIMER_OTVET.PT THEN
				STEP_INTO:=0;
				POPUTKA_PO_VREMENI_AVARIA:=POPUTKA_PO_VREMENI_AVARIA+1;
				TIMER_OTVET(IN:=FALSE, PT:=T#0s );
				TIMER_OTVET;
			END_IF
END_CASE
END_ACTION
ACTION SMS_AT_CMGS:
(*---------------------------------------------------------------------------------------------------AT+CMGS="ТЕЛЕФОННЫЙ НОМЕР"*)
CASE STEP_INTO OF
		0:
			STR_OK:='';
			STR_ERROR:='';
			OTVET:='';
			COMMAND:='';
			STEP_INTO:=1;
			TIMER_OTVET(IN:=FALSE, PT:=T#0s );
			TIMER_OTVET;
			PAUSA(IN:=FALSE, PT:=T#0s );
			PAUSA;
		1:
			COMMAND:='AT+CMGS="';(*<-------------------------------------------------------------------------------AT-КОМАНДА*)
			COMMAND:=CONCAT(COMMAND,number);
			COMMAND:=CONCAT(COMMAND,'"');
			STR_OK:='>';(*<--------------------------------------------------------------------------------------ПРАВИЛЬНЫЙ ОТВЕТ*)
			STR_ERROR:='ERROR';(*<-------------------------------------------------------------------------НЕПРАВИЛЬНЫЙ ОТВЕТ*)
			COMMAND:=CONCAT(COMMAND,'$R$N');
			SetByte(0,COMMAND,LEN(COMMAND));
			STEP_INTO:=2;
		2:
			FIND_OK:=FIND(OTVET, STR_OK);
			FIND_ERROR:=FIND(OTVET, STR_ERROR);

			IF FIND_OK<>0 THEN
				PAUSA(IN:=TRUE, PT:=ZADERGKA_PEREHODA );
				IF PAUSA.ET=PAUSA.PT THEN
					STEP_AVARIA:=70;(*<-------------------------------------------------ПЕРЕХОД К СЛЕДУЮЩЕЙ КОМАНДЕ*)(*70*)
					STEP_INTO:=0;
					POPUTKA_AVARIA:=0;
					POPUTKA_PO_VREMENI_AVARIA:=0;
				END_IF
			END_IF
			IF FIND_ERROR<>0 THEN
				STEP_INTO:=0;
				POPUTKA_AVARIA:=POPUTKA_AVARIA+1;
			END_IF
			TIMER_OTVET(IN:=TRUE, PT:=OGIDANIE_OTVETA );
			IF TIMER_OTVET.ET=TIMER_OTVET.PT THEN
				STEP_INTO:=0;
				POPUTKA_PO_VREMENI_AVARIA:=POPUTKA_PO_VREMENI_AVARIA+1;
				TIMER_OTVET(IN:=FALSE, PT:=T#0s );
				TIMER_OTVET;
			END_IF
END_CASE
END_ACTION
ACTION SMS_AT_CSCS_GSM:
(*--------------------------------------------------------------------------------------------------AT+CSCS="GSM" КОДИРОВКА GSM*)
CASE STEP_INTO OF
		0:
			STR_OK:='';
			STR_ERROR:='';
			OTVET:='';
			COMMAND:='';
			STEP_INTO:=1;
			TIMER_OTVET(IN:=FALSE, PT:=T#0s );
			TIMER_OTVET;
			PAUSA(IN:=FALSE, PT:=T#0s );
			PAUSA;
		1:
			COMMAND:='AT+CSCS="GSM"';(*<--------------------------------------------------------------------------AT-КОМАНДА*)
			STR_OK:='OK';(*<------------------------------------------------------------------------------------ПРАВИЛЬНЫЙ ОТВЕТ*)
			STR_ERROR:='ERROR';(*<-------------------------------------------------------------------------НЕПРАВИЛЬНЫЙ ОТВЕТ*)
			COMMAND:=CONCAT(COMMAND,'$R$N');
			SetByte(0,COMMAND,LEN(COMMAND));
			STEP_INTO:=2;
		2:
			FIND_OK:=FIND(OTVET, STR_OK);
			FIND_ERROR:=FIND(OTVET, STR_ERROR);

			IF FIND_OK<>0 THEN
				PAUSA(IN:=TRUE, PT:=ZADERGKA_PEREHODA );
				IF PAUSA.ET=PAUSA.PT THEN
					STEP_AVARIA:=60;(*<------------------------------------------------ПЕРЕХОД К СЛЕДУЮЩЕЙ КОМАНДЕ*)(*60*)
					STEP_INTO:=0;
					POPUTKA_AVARIA:=0;
					POPUTKA_PO_VREMENI_AVARIA:=0;
				END_IF
			END_IF
			IF FIND_ERROR<>0 THEN
				STEP_INTO:=0;
				POPUTKA_AVARIA:=POPUTKA_AVARIA+1;
			END_IF
			TIMER_OTVET(IN:=TRUE, PT:=OGIDANIE_OTVETA );
			IF TIMER_OTVET.ET=TIMER_OTVET.PT THEN
				STEP_INTO:=0;
				POPUTKA_PO_VREMENI_AVARIA:=POPUTKA_PO_VREMENI_AVARIA+1;
				TIMER_OTVET(IN:=FALSE, PT:=T#0s );
				TIMER_OTVET;
			END_IF
END_CASE
END_ACTION
ACTION SMS_ATE0:
(*----------------------------------------------------------------------------------------------------------------ATE0 ОТКЛЮЧИТЬ ЭХО*)
CASE STEP_INTO OF
		0:
			STR_OK:='';
			STR_ERROR:='';
			OTVET:='';
			COMMAND:='';
			STEP_INTO:=1;
			TIMER_OTVET(IN:=FALSE, PT:=T#0s );
			TIMER_OTVET;
			PAUSA(IN:=FALSE, PT:=T#0s );
			PAUSA;
		1:
			COMMAND:='ATE0';(*<--------------------------------------------------------------------------------------AT-КОМАНДА*)
			STR_OK:='OK'; (*<-----------------------------------------------------------------------------------ПРАВИЛЬНЫЙ ОТВЕТ*)
			STR_ERROR:='ERROR'; (*<------------------------------------------------------------------------НЕПРАВИЛЬНЫЙ ОТВЕТ*)
			COMMAND:=CONCAT(COMMAND,'$R$N');
			SetByte(0,COMMAND,LEN(COMMAND));
			STEP_INTO:=2;
		2:
			FIND_OK:=FIND(OTVET, STR_OK);
			FIND_ERROR:=FIND(OTVET, STR_ERROR);

			IF FIND_OK<>0 THEN
				PAUSA(IN:=TRUE, PT:=ZADERGKA_PEREHODA );
				IF PAUSA.ET=PAUSA.PT THEN
					STEP_AVARIA:=20;(*<-------------------------------------------------ПЕРЕХОД К СЛЕДУЮЩЕЙ КОМАНДЕ*)(*20*)
					STEP_INTO:=0;
					POPUTKA_AVARIA:=0;
					POPUTKA_PO_VREMENI_AVARIA:=0;
				END_IF
			END_IF
			IF FIND_ERROR<>0 THEN
				STEP_INTO:=0;
				POPUTKA_AVARIA:=POPUTKA_AVARIA+1;
			END_IF
			TIMER_OTVET(IN:=TRUE, PT:=OGIDANIE_OTVETA );
			IF TIMER_OTVET.ET=TIMER_OTVET.PT THEN
				STEP_INTO:=0;
				POPUTKA_PO_VREMENI_AVARIA:=POPUTKA_PO_VREMENI_AVARIA+1;
				TIMER_OTVET(IN:=FALSE, PT:=T#0s );
				TIMER_OTVET;
			END_IF
END_CASE
END_ACTION
ACTION SMS_SEND_DATA:
(*-------------------------------------------------------------------------------------------------------------------ПЕРЕДАЧА ДАННЫХ*)
CASE STEP_INTO OF
		0:
			STR_OK:='';
			STR_ERROR:='';
			OTVET:='';
			TIMER_OTVET(IN:=FALSE, PT:=T#0s );
			TIMER_OTVET;
			PAUSA(IN:=FALSE, PT:=T#0s );
			PAUSA;
			STRING_SEND:='';
			STRING_SEND_2:='';
			OTVET:='';
			STEP_INTO:=1;
		1:
			STR_OK:='+CMGS:';(*<-------------------------------------------------------------------------------ПРАВИЛЬНЫЙ ОТВЕТ*)
			STR_ERROR:='ERROR';(*<-------------------------------------------------------------------------НЕПРАВИЛЬНЫЙ ОТВЕТ*)
			STRING_SEND:='';
			STRING_SEND:=CONCAT(STRING_SEND,'KARAUL INGAVINO$R$N');
			MODEM_FORMIROVANIE_SMS_AVARII;(*------------------------------------ЗДЕСЬ ФОРМИРУЕТСЯ  СМС СООБЩЕНИЕ*)
			STRING_SEND:=CONCAT(STRING_SEND,'$R$N$R$N$1A$R$N');
			SetByte(0,STRING_SEND,LEN(STRING_SEND));

			OTVET:='';
			STR_FIND:=0;
			STEP_INTO:=2;
		2:
			FIND_OK:=FIND(OTVET, STR_OK);
			FIND_ERROR:=FIND(OTVET, STR_ERROR);

			IF FIND_OK<>0 THEN
				PAUSA(IN:=TRUE, PT:=ZADERGKA_PEREHODA );
				IF PAUSA.ET=PAUSA.PT THEN
					STEP_INTO:=3;
					POPUTKA_AVARIA:=0;
					POPUTKA_PO_VREMENI_AVARIA:=0;
				END_IF
			END_IF
			IF FIND_ERROR<>0 THEN
				PAUSA(IN:=TRUE, PT:=ZADERGKA_PEREHODA );
				IF PAUSA.ET=PAUSA.PT THEN
					STEP_INTO:=3;
				END_IF
			END_IF
			TIMER_OTVET(IN:=TRUE, PT:=OGIDANIE_OTVETA );
			IF TIMER_OTVET.ET=TIMER_OTVET.PT THEN
				POPUTKA_PO_VREMENI_AVARIA:=POPUTKA_PO_VREMENI_AVARIA+1;
				TIMER_OTVET(IN:=FALSE, PT:=T#0s );
				TIMER_OTVET;
			END_IF
		3:

			STR_OK:='';
			STR_ERROR:='';
			STR_OK:='OK';(*<------------------------------------------------------------------------------------ПРАВИЛЬНЫЙ ОТВЕТ*)
			STR_ERROR:='ERROR';(*<-------------------------------------------------------------------------НЕПРАВИЛЬНЫЙ ОТВЕТ*)
			TIMER_OTVET(IN:=FALSE, PT:=T#0s );
			TIMER_OTVET;
			PAUSA(IN:=FALSE, PT:=T#0s );
			PAUSA;
			STEP_INTO:=4;
		4:
			FIND_OK:=FIND(OTVET, STR_OK);
			FIND_ERROR:=FIND(OTVET, STR_ERROR);

			IF FIND_OK<>0 THEN
				PAUSA(IN:=TRUE, PT:=ZADERGKA_PEREHODA );
				IF PAUSA.ET=PAUSA.PT THEN
					TEL:=TEL+1;
					IF TEL>KOLICHESTVO_NOMEROV THEN
						TEL:=1;
					END_IF
					STEP_AVARIA:=75;(*<-------------------------------------------------ПЕРЕХОД К СЛЕДУЮЩЕЙ КОМАНДЕ*)(*75*)
					STEP_INTO:=0;
					POPUTKA_AVARIA:=0;
					POPUTKA_PO_VREMENI_AVARIA:=0;
				END_IF
			END_IF
			IF FIND_ERROR<>0 THEN
				PAUSA(IN:=TRUE, PT:=ZADERGKA_PEREHODA );
				IF PAUSA.ET=PAUSA.PT THEN
					STEP_AVARIA:=75;(*<------------------------------------------------ПЕРЕХОД К СЛЕДУЮЩЕЙ КОМАНДЕ*)(*75*)
					STEP_INTO:=0;
					POPUTKA_AVARIA:=0;
					POPUTKA_PO_VREMENI_AVARIA:=0;
				END_IF
			END_IF
			TIMER_OTVET(IN:=TRUE, PT:=OGIDANIE_OTVETA );
			IF TIMER_OTVET.ET=TIMER_OTVET.PT THEN
				STEP_INTO:=3;
				POPUTKA_PO_VREMENI_AVARIA:=POPUTKA_PO_VREMENI_AVARIA+1;
				TIMER_OTVET(IN:=FALSE, PT:=T#0s );
				TIMER_OTVET;
			END_IF
	END_CASE
END_ACTION

(* POU GORELKA_PROGRESSIVNAYA, ST *)
FUNCTION_BLOCK GORELKA_PROGRESSIVNAYA
VAR_INPUT
	PUSK:BOOL; (*---------------------------------------------------------------------------------------------------ПУСК ГОРЕЛКИ*)
	TEMPERATURA_KOTLA:REAL; (*-----------------------------------------------------------ТЕМПЕРАТУРА НА ВЫХОДЕ КОТЛА*)
	TEMPERATURA_POROG_1:REAL; (*-----------------------------------------------1 ПОРОГ. ОТКЛЮЧЕНИЕ ВТОРОЙ СТУПЕНИ*)
	TEMPERATURA_POROG_2:REAL; (*----------------------------------------------------2 ПОРОГ. ОТКЛЮЧЕНИЕ ТЕРМОСТАТА*)
	TEMPERATURA_POROG_3:REAL; (*------------------------------------------ТЕМПЕРАТУРА ДО КОТОРОЙ ОСТЫВАЕТ КОТЕЛ*)
	GISTEREZIS:REAL;(*----------------------------------------------------------------ГИСТЕРЕЗИС ПЕРЕКЛЮЧЕНИЯ 2 СТУПЕНИ*)
	S3:BOOL; (*----------------------------------------------------------------ОШИБКА. ПРИЛЕТАЕТ С КОТЛА. 220 В ЧЕРЕЗ РЕЛЕ*)
	B4:BOOL; (*----------------------------------------------------------------РАБОТА. ПРИЛЕТАЕТ С КОТЛА. 220 В ЧЕРЕЗ РЕЛЕ*)
	SBROS_ERROR:BOOL;(*----------------------------------------------------------------------------------------СБРОС ОШИБКИ*)
	TIME_SBROS_ERROR:TIME;(*----------------------------------------------------------ВРЕМЯ НУЖНОЕ ДЛЯ СБРОСА АВАРИИ*)
END_VAR
VAR_IN_OUT
	ERROR:BOOL;(*----------------------------------------------------------------------------------------------------------АВАРИЯ*)
END_VAR
VAR_OUTPUT
	T1_T2:BOOL; (*----------------------------------------------------------------------------------КЛЕММЫ ЗАПРОС НА РОЗЖИГ*)
	TMIN_TMAX:BOOL; (*-------------------------------------------------------------------КЛЕММЫ БОЛЬШОЕ/МАЛОЕ ГОРЕНИЕ*)
	WORK:BOOL;(*--------------------------------------------------------------------------------------СТАТУС РАБОТЫ ГОРЕЛКИ*)
END_VAR
VAR
	MASTER:BYTE:=0;
	STEP_SBROS_ERROR:BYTE:=0;
	STEP:INT:=0;
	TIMER:TP;
END_VAR
IF S3=TRUE THEN(*---ЕСЛИ ПРИЛЕТАЕТ ОШИБКА 220 В С РЕЛЕ ТО НЕ ВКЮЧАЕМ ГОРЕЛКУ , В ПАМЯТЬ ЗПИСЫВАЕМ ОШИБКУ*)
	ERROR:=TRUE;
	WORK:=FALSE;
	PUSK:=FALSE;
END_IF

IF ERROR=FALSE THEN(*----------------------------------------------------------------------------ЕСЛИ В ПАМЯТИ НЕТ ОШИБОК*)
	IF PUSK=TRUE THEN(*----------------------------------------------ЗАПУСК ФУНКЦИОНАЛЬНОГО БЛОКА РАБОТЫ ГОРЕЛКИ*)
		CASE MASTER OF
			0:
				T1_T2:=TRUE;
				MASTER:=1;
			1:
				IF S3=FALSE THEN (*----------------------------------------------------------ЕСЛИ НЕТ ОШИБКИ 220 С ГОРЕЛКИ*)
					IF B4 THEN (*--------------------------------------------ЕСЛИ ГОРЕЛКА РАБОТАЕТ, ПРИЛЕТЕЛО 220 С РЕЛЕ*)
						CASE STEP OF
							0:
								IF 	TEMPERATURA_KOTLA<TEMPERATURA_POROG_1 THEN (*---------------МЕНЬШЕ 1 ПОРОГА*)
									TMIN_TMAX:=TRUE;
								END_IF
								IF	TEMPERATURA_KOTLA>=TEMPERATURA_POROG_1
																	AND TEMPERATURA_KOTLA< TEMPERATURA_POROG_2 THEN
									TMIN_TMAX:=FALSE;(*------------------------------БОЛЬШЕ 1 ПОРОГА И МЕНЬШЕ 2 ПОРОГА*)
									STEP:=1;
								END_IF
								IF	TEMPERATURA_KOTLA>TEMPERATURA_POROG_2 THEN
									T1_T2:=FALSE;
									TMIN_TMAX:=FALSE;
									MASTER:=3;
								END_IF
							1:(*-----------------------------------------------------------ЕСЛИ МЕНЬШЕ 1 ПОРОГА - ГИСТЕРЕЗИС*)
								IF 	TEMPERATURA_KOTLA<TEMPERATURA_POROG_1-GISTEREZIS THEN
									STEP:=0;
								END_IF
								IF	TEMPERATURA_KOTLA>TEMPERATURA_POROG_2 THEN
									T1_T2:=FALSE;
									TMIN_TMAX:=FALSE;
									MASTER:=3;
								END_IF
						END_CASE
					ELSE
						MASTER:=0;
					END_IF
				ELSE
					MASTER:=2;
				END_IF
			2:
				ERROR:=TRUE;
				PUSK:=FALSE;
				T1_T2:=FALSE;
				TMIN_TMAX:=FALSE;
			3:
				IF TEMPERATURA_KOTLA<TEMPERATURA_POROG_3 THEN (*остывание*)
					MASTER:=0;
				END_IF
		END_CASE
	ELSE
		T1_T2:=FALSE;
		TMIN_TMAX:=FALSE;
		MASTER:=0;
	END_IF
ELSE  (*----------------------------------------------------------------------------------------------ЕСЛИ  В ПАМЯТИ НЕТ ОШИБОК*)
	PUSK:=FALSE;
	T1_T2:=FALSE;
	TMIN_TMAX:=FALSE;
	MASTER:=0;
END_IF


IF S3=FALSE AND ERROR=FALSE AND PUSK=TRUE AND B4=TRUE THEN(*----ЕСЛИ НЕТ ОШИБКИ 220В,  НЕТ ОШИБКИ В ПАМЯТИ*)
	WORK:=TRUE;(*-----------------------------------------------------------------------ПУСК И РАБОТА 220 ТО, СТАТУС РАБОТА*)
END_IF
IF PUSK=FALSE OR S3 OR ERROR THEN
	WORK:=FALSE;(*---------------------------------------------------------------------НЕ ПУСК ИЛИ АВАРИЯ, СТАТУС НЕ РАБОТА*)
END_IF
(*----------------------------------------------------------------------СБРОС ОШИБКИ И ВРЕМЯ ДЛЯ СБРОСА НА САМОЙ ГОРЕЛКЕ*)
IF SBROS_ERROR=TRUE  THEN
	STEP_SBROS_ERROR:=1;
END_IF
CASE STEP_SBROS_ERROR OF
	1:
		ERROR := FALSE;
		T1_T2:=TRUE;
		TIMER(IN:=TRUE, PT:=TIME_SBROS_ERROR);
		IF  TIMER.ET=TIMER.PT THEN
			MASTER:=0;
			SBROS_ERROR:=FALSE;
			PUSK:=TRUE;
			T1_T2:=FALSE;
			STEP_SBROS_ERROR:=0;
			TIMER(IN:=FALSE,PT:=T#0s);
      		 	TIMER;
		END_IF
END_CASE
END_FUNCTION_BLOCK

(* POU KASKAD_1_NASOS_1_DATCHIKA_DAVLENIA, ST *)
FUNCTION_BLOCK KASKAD_1_NASOS_1_DATCHIKA_DAVLENIA
VAR
	TP1: TP; (*--------------------------------------------------------------------------------------ПАУЗА ДЛЯ ПЕРЕПАДА ДАВЛЕНИЯ*)
	STEP:BYTE:=0; (*------------------------------------------------------------------------------------------СТАДИЯ ВЫПОЛНЕНИЯ*)
	STEP1:BYTE:=0; (*--------------------------------------------------------------------КРАТКОВРЕМЕННОЕ ПАДЕНИЕ ДАВЛЕНИЯ*)
	DELTA_P:REAL; (*-----------------------------------------------------------------------------------РАЗНИЦА ДАВЛЕНИЙ P1 и P2*)
END_VAR
VAR_INPUT
	TIME_AVARIA:TIME;(*-----------------------------------------------------------------------------------------ВРЕМЯ НА АВАРИЮ*)
	P_1:REAL; (*------------------------------------------------------------------------------------------ДАВЛЕНИЕ ПОСЛЕ КАСКАДА*)
	P_USTAVKA:REAL; (*-------------------------------------------------------------------------УСТАВКА НИЖЕ КОТОРОЙ АВАРИЯ*)
	SBROS_ERROR: BOOL; (*------------------------------------------------------------------СБРОС ОШИБКИ КАСКАДА НАСОСОВ*)
	PUSK_NASOS:BOOL; (*--------------------------------------------------------------------------------ПУСК КАСКАДА НАСОСОВ*)
END_VAR
VAR_IN_OUT
	ERROR_NASOS1: BOOL; (*-------------------------------------------ОШИБКА НАСОСА 1. ХРАНИТСЯ В RETAIN КОНТРОЛЛЕРА*)
END_VAR
VAR_OUTPUT
	RELE_NASOS1:BOOL; (*-----------------------------------------------------------------------------РЕЛЕ ВКЛЮЧЕНИЯ НАСОСА 1*)
	WORK:BOOL;(*-----------------------------------------------------------------------------СТАТУС РАБОТА КАСКАДА НАСОСОВ*)
END_VAR
IF SBROS_ERROR=TRUE  THEN(*----------------------------------------СБРОС КАСКАДА НАСОСОВ, И ОБНУЛЕНИЕ ПАРАМЕТРОВ*)
	ERROR_NASOS1:= FALSE;
	STEP:=0;
	STEP1:=0;
	SBROS_ERROR:=FALSE;
END_IF



IF ERROR_NASOS1=TRUE THEN(*------------------------------------ЕСЛИ ОШИБКА НА ДВУХ НАСОСАХ, ТО ВЫКЛЮЧИТЬ КАСКАД*)
	PUSK_NASOS:=FALSE;
END_IF


IF PUSK_NASOS=TRUE THEN(*---------------------------------------------------ЕСЛИ ДАНА КОМАНДА ПУСК КАСКАДА НАСОСОВ*)

	IF ERROR_NASOS1=FALSE  THEN(*-----------------------------------------------ЕСЛИ НА ОДНОМ ИЗ НАСОСОВ НЕТ ОШИБКИ*)
		CASE STEP OF
			0:
				IF ERROR_NASOS1=TRUE THEN STEP:=2;(*----------------ЕСЛИ ОШИБКА 1 НАСОСА, ВКЛЮЧАЕМ СРАЗУ ВТОРОЙ*)
             			ELSE
 					RELE_NASOS1:=1;
					STEP:=1;
				END_IF
			1:
				IF P_1<P_USTAVKA THEN	(*--ЕСЛИ ПЕРЕПАД ДАВЛЕНИЯ < УСТАВКИ ТО НАЧИНАЕМ ОСЧЕТ В СЕК.*)
   				CASE STEP1 OF
					0:
						TP1(IN:=TRUE,PT:=TIME_AVARIA);
						IF  TP1.ET=TP1.PT THEN
							STEP1:=1;
							TP1(IN:=FALSE,PT:=T#0s);
      		 					TP1;
						END_IF
					1:
						IF  (ERROR_NASOS1=TRUE)  OR (P_1<P_USTAVKA)  THEN
							RELE_NASOS1:=0;
							ERROR_NASOS1:=TRUE;
							STEP1:=0;
							STEP:=2;
						ELSE
							STEP1:=0;
						END_IF
				END_CASE
				ELSE
					TP1(IN:=FALSE,PT:=T#0s);
      		 			TP1;
				END_IF
			2:
				RELE_NASOS1:=0;
		END_CASE
	END_IF(*----------------------------------------------------------------------------ЕСЛИ НА ОДНОМ ИЗ НАСОСОВ НЕТ ОШИБКИ*)
ELSE(*-----------------------------------------------------------------------------ЕСЛИ ДАНА КОМАНДА ПУСК КАСКАДА НАСОСОВ*)
	RELE_NASOS1:=0;
	STEP:=0;
	STEP1:=0;(*--------------------------------------ДОБАВИЛ ОБНУЛЕНИЕ ВСЛЕПУЮ, НАДО ПРОВЕРИТЬ НУЖНО ЛИ ОНО ЗДЕСЬ*)
	TP1(IN:=FALSE,PT:=T#0s);
	TP1;
END_IF


(*---------------------------------------------ЕСЛИ 1 ИЛИ 2 НАСОС ВКЛЮЧЕН И ПУСК КАСКАДА ТО СТАТУС КАСКАДА "РАБОТА"*)
IF (RELE_NASOS1=1) AND (PUSK_NASOS=TRUE) THEN WORK:=TRUE; END_IF
(*---------------------------ЕСЛИ 1 И 2 НАСОС ВЫКЛЮЧЕНЫ И ПУСК КАСКАДА ВЫКЛЮЧЕН ТО СТАТУС КАСКАДА "НЕТ РАБОТЫ"*)
IF (RELE_NASOS1=0) AND (PUSK_NASOS=FALSE) THEN WORK:=FALSE; END_IF
END_FUNCTION_BLOCK

(* POU KASKAD_1_NASOS_2_DATCHIKA_DAVLENIA, ST *)
FUNCTION_BLOCK KASKAD_1_NASOS_2_DATCHIKA_DAVLENIA
VAR
	TP1: TP; (*--------------------------------------------------------------------------------------ПАУЗА ДЛЯ ПЕРЕПАДА ДАВЛЕНИЯ*)
	STEP:BYTE:=0; (*------------------------------------------------------------------------------------------СТАДИЯ ВЫПОЛНЕНИЯ*)
	STEP1:BYTE:=0; (*--------------------------------------------------------------------КРАТКОВРЕМЕННОЕ ПАДЕНИЕ ДАВЛЕНИЯ*)
	DELTA_P:REAL; (*-----------------------------------------------------------------------------------РАЗНИЦА ДАВЛЕНИЙ P1 и P2*)
END_VAR
VAR_INPUT
	TIME_AVARIA:TIME;(*-----------------------------------------------------------------------------------------ВРЕМЯ НА АВАРИЮ*)
	P_1:REAL; (*------------------------------------------------------------------------------------------ДАВЛЕНИЕ ПОСЛЕ КАСКАДА*)
	P_2:REAL; (*----------------------------------------------------------------------------------------ДАВЛЕНИЕ ПЕРЕД КАСКАДОМ*)
	PEREPAD_DAVLENIA:REAL; (*-------------------------------------------------------------------------------ПЕРЕПАД ДАВЛЕНИЯ*)
	SBROS_ERROR: BOOL; (*------------------------------------------------------------------СБРОС ОШИБКИ КАСКАДА НАСОСОВ*)
	PUSK_NASOS:BOOL; (*--------------------------------------------------------------------------------ПУСК КАСКАДА НАСОСОВ*)
END_VAR
VAR_IN_OUT
	ERROR_NASOS1: BOOL; (*-------------------------------------------ОШИБКА НАСОСА 1. ХРАНИТСЯ В RETAIN КОНТРОЛЛЕРА*)
END_VAR
VAR_OUTPUT
	RELE_NASOS1:BOOL; (*-----------------------------------------------------------------------------РЕЛЕ ВКЛЮЧЕНИЯ НАСОСА 1*)
	WORK:BOOL;(*-----------------------------------------------------------------------------СТАТУС РАБОТА КАСКАДА НАСОСОВ*)
END_VAR
IF SBROS_ERROR=TRUE  THEN(*----------------------------------------СБРОС КАСКАДА НАСОСОВ, И ОБНУЛЕНИЕ ПАРАМЕТРОВ*)
	ERROR_NASOS1:= FALSE;
	STEP:=0;
	STEP1:=0;
	SBROS_ERROR:=FALSE;
END_IF

DELTA_P:=P_1-P_2;(*---------------------------------------------------------------------------------РАСЧЕТ ПЕРЕПАДА ДАВЛЕНИЯ *)

IF ERROR_NASOS1=TRUE THEN(*------------------------------------ЕСЛИ ОШИБКА НА ДВУХ НАСОСАХ, ТО ВЫКЛЮЧИТЬ КАСКАД*)
	PUSK_NASOS:=FALSE;
END_IF


IF PUSK_NASOS=TRUE THEN(*---------------------------------------------------ЕСЛИ ДАНА КОМАНДА ПУСК КАСКАДА НАСОСОВ*)

	IF ERROR_NASOS1=FALSE  THEN(*-----------------------------------------------ЕСЛИ НА ОДНОМ ИЗ НАСОСОВ НЕТ ОШИБКИ*)
		CASE STEP OF
			0:
				IF ERROR_NASOS1=TRUE THEN STEP:=2;(*----------------ЕСЛИ ОШИБКА 1 НАСОСА, ВКЛЮЧАЕМ СРАЗУ ВТОРОЙ*)
             			ELSE
 					RELE_NASOS1:=1;
					STEP:=1;
				END_IF
			1:
				IF DELTA_P<PEREPAD_DAVLENIA THEN	(*--ЕСЛИ ПЕРЕПАД ДАВЛЕНИЯ < УСТАВКИ ТО НАЧИНАЕМ ОСЧЕТ В СЕК.*)
   				CASE STEP1 OF
					0:
						TP1(IN:=TRUE,PT:=TIME_AVARIA);
						IF  TP1.ET=TP1.PT THEN
							STEP1:=1;
							TP1(IN:=FALSE,PT:=T#0s);
      		 					TP1;
						END_IF
					1:
						IF  (ERROR_NASOS1=TRUE)  OR (DELTA_P<PEREPAD_DAVLENIA)  THEN
							RELE_NASOS1:=0;
							ERROR_NASOS1:=TRUE;
							STEP1:=0;
							STEP:=2;
						ELSE
							STEP1:=0;
						END_IF
				END_CASE
				ELSE
					TP1(IN:=FALSE,PT:=T#0s);
      		 			TP1;
				END_IF
			2:
				RELE_NASOS1:=0;
		END_CASE
	END_IF(*----------------------------------------------------------------------------ЕСЛИ НА ОДНОМ ИЗ НАСОСОВ НЕТ ОШИБКИ*)
ELSE(*-----------------------------------------------------------------------------ЕСЛИ ДАНА КОМАНДА ПУСК КАСКАДА НАСОСОВ*)
	RELE_NASOS1:=0;
	STEP:=0;
	STEP1:=0;(*--------------------------------------ДОБАВИЛ ОБНУЛЕНИЕ ВСЛЕПУЮ, НАДО ПРОВЕРИТЬ НУЖНО ЛИ ОНО ЗДЕСЬ*)
	TP1(IN:=FALSE,PT:=T#0s);
	TP1;
END_IF


(*---------------------------------------------ЕСЛИ 1 ИЛИ 2 НАСОС ВКЛЮЧЕН И ПУСК КАСКАДА ТО СТАТУС КАСКАДА "РАБОТА"*)
IF (RELE_NASOS1=1) AND (PUSK_NASOS=TRUE) THEN WORK:=TRUE; END_IF
(*---------------------------ЕСЛИ 1 И 2 НАСОС ВЫКЛЮЧЕНЫ И ПУСК КАСКАДА ВЫКЛЮЧЕН ТО СТАТУС КАСКАДА "НЕТ РАБОТЫ"*)
IF (RELE_NASOS1=0) AND (PUSK_NASOS=FALSE) THEN WORK:=FALSE; END_IF
END_FUNCTION_BLOCK
